		// Properties:
		IF (BACnet_Param.bStateText_WriteProtect) THEN
			WriteProtectProperty(E_BACnetPropIdentifier.PropActiveText, TRUE);
			WriteProtectProperty(E_BACnetPropIdentifier.PropInactiveText, TRUE);
		END_IF
		
		// Ensure UTF-8 Encoding:
		F_BA_EnsureUTF8(ADR(sDeviceType), SIZEOF(sDeviceType));
		F_BA_EnsureUTF8(ADR(sInactiveText), SIZEOF(sInactiveText));
		F_BA_EnsureUTF8(ADR(sActiveText), SIZEOF(sActiveText));

	TCOM_STATE.TCOM_STATE_SAFEOP:
		SyncPropertyPvPrio(E_BACnetPropIdentifier.PropPresentValue, SIZEOF(bValPgm), ADR(bValPgm), ADR(bEnPgm), BACnet_Param.ePrio_Program, 0, eFullSync_InitPLC, TRUE);
		
		SyncProperty(E_BACnetPropIdentifier.PropPresentValue, SIZEOF(bPresentValue), ADR(bPresentValue), 0, eSync_FromSupplement, TRUE);
		SyncProperty(E_BACnetPropIdentifier.PropCurrentlyActivePriority, SIZEOF(eActivePrio), ADR(eActivePrio), 0, eSync_FromSupplement, TRUE);
		
		SyncProperty(E_BACnetPropIdentifier.PropFeedbackValue, SIZEOF(_bFeedbackValue), ADR(_bFeedbackValue), 0, eSync_ToSupplement, TRUE);
		
	TCOM_STATE.TCOM_STATE_OP:
		SyncProperty(E_BACnetPropIdentifier.PropDeviceType, SIZEOF(sDeviceType), ADR(sDeviceType), 0, eFullSync_InitPLC, FALSE);
		SyncProperty(E_BACnetPropIdentifier.PropOutOfService, SIZEOF(bOutOfService), ADR(bOutOfService), 0, eFullSync_InitPLC, FALSE);
		SyncProperty(E_BACnetPropIdentifier.PropMinimumOffTime, SIZEOF(nMinimumOffTime), ADR(nMinimumOffTime), 0, eFullSync_InitPLC, FALSE);	
		SyncProperty(E_BACnetPropIdentifier.PropMinimumOnTime, SIZEOF(nMinimumOnTime), ADR(nMinimumOnTime), 0, eFullSync_InitPLC, FALSE);	
		SyncProperty(E_BACnetPropIdentifier.PropRelinquishDefault, SIZEOF(bRelinquishDefault), ADR(bRelinquishDefault), 0, eFullSync_InitPLC, FALSE);	
		SyncProperty(E_BACnetPropIdentifier.PropActiveText, SIZEOF(sActiveText), ADR(sActiveText), 0, eFullSync_InitPLC, FALSE);	
		SyncProperty(E_BACnetPropIdentifier.PropInactiveText, SIZEOF(sInactiveText), ADR(sInactiveText), 0, eFullSync_InitPLC, FALSE);
		SyncProperty(E_BACnetPropIdentifier.PropPolarity, SIZEOF(ePolarity), ADR(ePolarity), 0, eFullSync_InitPLC, FALSE);

		SyncProperty(E_BACnetPropIdentifier.PropChangeOfStateCount, SIZEOF(nChangeOfStateCount), ADR(nChangeOfStateCount), 0, eFullSync_InitPLC, FALSE);
		SyncProperty(E_BACnetPropIdentifier.PropChangeOfStateTime, SIZEOF(stChangeOfStateTime), ADR(stChangeOfStateTime), 0, eSync_FromSupplement, FALSE);
		SyncProperty(E_BACnetPropIdentifier.PropTimeOfStateCountReset, SIZEOF(stTimeOfStateCountReset), ADR(stTimeOfStateCountReset), 0, eSync_FromSupplement, FALSE);

		SyncProperty(E_BACnetPropIdentifier.PropElapsedActiveTime, SIZEOF(nElapsedActiveTime), ADR(nElapsedActiveTime), 0, eFullSync_InitPLC, FALSE);
		SyncProperty(E_BACnetPropIdentifier.PropTimeOfActiveTimeReset, SIZEOF(stTimeOfActiveTimeReset), ADR(stTimeOfActiveTimeReset), 0, eSync_FromSupplement, FALSE);
		
END_CASE
END_METHOD

METHOD FB_init : BOOL
VAR_INPUT
	bInitRetains : BOOL; // if TRUE, the retain variables are initialized (warm start / cold start)
	bInCopyCode : BOOL;  // if TRUE, the instance afterwards gets moved into the copy code (online change)
END_VAR
eObjectType := E_BACnetObjType.ObjBinaryOutput;
END_METHOD

PROPERTY ActivePrio : E_BACnet_Priority
GET
ActivePrio := eActivePrio;
END_GET
END_PROPERTY

PROPERTY ChangeOfStateTime : ST_BA_DateTime
GET
ChangeOfStateTime := stChangeOfStateTime;
END_GET
END_PROPERTY

PROPERTY TimeOfActiveTimeReset : ST_BA_DateTime
GET
TimeOfActiveTimeReset := stTimeOfActiveTimeReset;
END_GET
END_PROPERTY

PROPERTY TimeOfStateCountReset : ST_BA_DateTime
GET
TimeOfStateCountReset := stTimeOfStateCountReset;
END_GET
END_PROPERTY

END_FUNCTION_BLOCK

// POUs/Local/Objects/5P/FB_BACnet_BO_Raw5P
// Binary Output Object
// - Raw communication
// - 5 Priorities
{attribute 'pin_presentation_order_inputs' := 'bEnSfty,bValSfty,bEnCrit,bValCrit,bEnManLoc,bValManLoc,bEnPgm,bValPgm'}
{attribute 'pin_presentation_order_outputs' := 'bPresentValue,eActivePrio,bEvent,eReliability'}
{attribute 'enable_dynamic_creation'}
FUNCTION_BLOCK FB_BACnet_BO_Raw5P EXTENDS FB_BACnet_BO_Raw
VAR_INPUT
	bEnSfty					: BOOL;
	bValSfty				: BOOL;
	bEnCrit					: BOOL;
	bValCrit				: BOOL;
	bEnManLoc				: BOOL;
	bValManLoc				: BOOL;
END_VAR
VAR_INPUT CONSTANT PERSISTENT
	{region 'Operational Parameters'}
		{attribute 'parameterCategory':='Manual'}
		bEnManualRm : BOOL;
		{attribute 'parameterCategory':='Manual'}
		bValManualRm : BOOL;
	{endregion}
END_VAR

SUPER^();

METHOD PROTECTED OnObjectStateChanged
SUPER^.OnObjectStateChanged();

CASE (tState) OF
	TCOM_STATE.TCOM_STATE_PREOP:
		// SyncHandler:
		RequestSyncHandlers(1, 4);
		
	TCOM_STATE.TCOM_STATE_SAFEOP:
		SyncPropertyPvPrio(E_BACnetPropIdentifier.PropPresentValue, SIZEOF(bValSfty), ADR(bValSfty), ADR(bEnSfty), BACnet_Param.ePrio_LifeSafety, 0, eFullSync_InitPLC, TRUE);
		SyncPropertyPvPrio(E_BACnetPropIdentifier.PropPresentValue, SIZEOF(bValCrit), ADR(bValCrit), ADR(bEnCrit), BACnet_Param.ePrio_Critical, 0, eFullSync_InitPLC, TRUE);
		SyncPropertyPvPrio(E_BACnetPropIdentifier.PropPresentValue, SIZEOF(bValManLoc), ADR(bValManLoc), ADR(bEnManLoc), BACnet_Param.ePrio_ManLocal, 0, eFullSync_InitPLC, TRUE);
		SyncPropertyPvPrio(E_BACnetPropIdentifier.PropPresentValue, SIZEOF(bValManualRm), ADR(bValManualRm), ADR(bEnManualRm), BACnet_Param.ePrio_ManRemote, 0, eFullSync_InitPLC, TRUE);
		
	TCOM_STATE.TCOM_STATE_OP:
		;
		
END_CASE
END_METHOD

PROPERTY EnManualRm : BOOL
GET
EnManualRm := bEnManualRm;
END_GET
SET
bEnManualRm := EnManualRm;
END_SET
END_PROPERTY

PROPERTY ValManualRm : BOOL
GET
ValManualRm := bValManualRm;
END_GET
SET
bValManualRm := ValManualRm;
END_SET
END_PROPERTY

END_FUNCTION_BLOCK

// POUs/Local/Objects/FB_BACnet_BV
// Binary Value Object
// - 1 Priority
{attribute 'enable_dynamic_creation'}
FUNCTION_BLOCK FB_BACnet_BV EXTENDS FB_BACnet_EventObject
VAR_INPUT
	bEnPgm		: BOOL;
	bValPgm		: BOOL;
END_VAR
VAR_INPUT CONSTANT PERSISTENT
	{region 'Variable Parameters'}
		{attribute 'parameterCategory':='General'}
		{attribute 'parameterUnit':= 's'}
		nMinimumOffTime : UDINT;
		{attribute 'parameterCategory':='General'}
		{attribute 'parameterUnit':= 's'}
		nMinimumOnTime : UDINT;
		
		{attribute 'parameterCategory':='Value'}
		bRelinquishDefault : BOOL;
		{attribute 'parameterCategory':='Value'}
		bOutOfService : BOOL;
		{attribute 'parameterCategory':='Value'}
		{attribute 'TcEncoding':='UTF-8'}
		sInactiveText : T_BACnet_StateText;
		{attribute 'parameterCategory':='Value'}
		{attribute 'TcEncoding':='UTF-8'}
		sActiveText : T_BACnet_StateText;
		
		{attribute 'parameterCategory':='EventConfig'}
		bAlarmValue : BOOL := TRUE;
			 
		{attribute 'parameterCategory':='StateChange'}
		nChangeOfStateCount : UDINT;
		
		{attribute 'parameterCategory':='ActiveTime'}
		{attribute 'parameterUnit':= 's'}
		nElapsedActiveTime : UDINT;
	{endregion}
END_VAR
VAR_OUTPUT
	bPresentValue	: BOOL;
	eActivePrio		: E_BACnet_Priority;			// Indicates the currently active priority of the priority array
END_VAR
VAR
	{region 'Output-Properties'}
		{attribute 'parameterCategory':='StateChange'}
		stChangeOfStateTime : ST_BA_DateTime;
		{attribute 'parameterCategory':='StateChange'}
		stTimeOfStateCountReset : ST_BA_DateTime;
		
		{attribute 'parameterCategory':='ActiveTime'}
		stTimeOfActiveTimeReset : ST_BA_DateTime;
	{endregion}
END_VAR

SUPER^();

METHOD PROTECTED OnObjectStateChanged
SUPER^.OnObjectStateChanged();

CASE (tState) OF
	TCOM_STATE.TCOM_STATE_PREOP:
		// SyncHandler:
		RequestSyncHandlers(4, 10);
		
		// Properties:
		EnableProperty(E_BACnetPropIdentifier.PropDeviceType, FALSE);

		IF (BACnet_Param.bStateText_WriteProtect) THEN
			WriteProtectProperty(E_BACnetPropIdentifier.PropActiveText, TRUE);
			WriteProtectProperty(E_BACnetPropIdentifier.PropInactiveText, TRUE);
		END_IF
		
		// Ensure UTF-8 Encoding:
		F_BA_EnsureUTF8(ADR(sInactiveText), SIZEOF(sInactiveText));
		F_BA_EnsureUTF8(ADR(sActiveText), SIZEOF(sActiveText));

	TCOM_STATE.TCOM_STATE_SAFEOP:
		SyncPropertyPvPrio(E_BACnetPropIdentifier.PropPresentValue, SIZEOF(bValPgm), ADR(bValPgm), ADR(bEnPgm), BACnet_Param.ePrio_Program, 0, eFullSync_InitPLC, TRUE);
		
		SyncProperty(E_BACnetPropIdentifier.PropPresentValue, SIZEOF(bPresentValue), ADR(bPresentValue), 0, eSync_FromSupplement, TRUE);
		SyncProperty(E_BACnetPropIdentifier.PropCurrentlyActivePriority, SIZEOF(eActivePrio), ADR(eActivePrio), 0, eSync_FromSupplement, TRUE);
		
	TCOM_STATE.TCOM_STATE_OP:
		SyncProperty(E_BACnetPropIdentifier.PropAlarmValue, SIZEOF(bAlarmValue), ADR(bAlarmValue), 0, eFullSync_InitPLC, FALSE);
		SyncProperty(E_BACnetPropIdentifier.PropOutOfService, SIZEOF(bOutOfService), ADR(bOutOfService), 0, eFullSync_InitPLC, FALSE);
		SyncProperty(E_BACnetPropIdentifier.PropMinimumOffTime, SIZEOF(nMinimumOffTime), ADR(nMinimumOffTime), 0, eFullSync_InitPLC, FALSE);	
		SyncProperty(E_BACnetPropIdentifier.PropMinimumOnTime, SIZEOF(nMinimumOnTime), ADR(nMinimumOnTime), 0, eFullSync_InitPLC, FALSE);	
		SyncProperty(E_BACnetPropIdentifier.PropRelinquishDefault, SIZEOF(bRelinquishDefault), ADR(bRelinquishDefault), 0, eFullSync_InitPLC, FALSE);	
		SyncProperty(E_BACnetPropIdentifier.PropActiveText, SIZEOF(sActiveText), ADR(sActiveText), 0, eFullSync_InitPLC, FALSE);	
		SyncProperty(E_BACnetPropIdentifier.PropInactiveText, SIZEOF(sInactiveText), ADR(sInactiveText), 0, eFullSync_InitPLC, FALSE);

		SyncProperty(E_BACnetPropIdentifier.PropChangeOfStateCount, SIZEOF(nChangeOfStateCount), ADR(nChangeOfStateCount), 0, eFullSync_InitPLC, FALSE);
		SyncProperty(E_BACnetPropIdentifier.PropChangeOfStateTime, SIZEOF(stChangeOfStateTime), ADR(stChangeOfStateTime), 0, eSync_FromSupplement, FALSE);
		SyncProperty(E_BACnetPropIdentifier.PropTimeOfStateCountReset, SIZEOF(stTimeOfStateCountReset), ADR(stTimeOfStateCountReset), 0, eSync_FromSupplement, FALSE);

		SyncProperty(E_BACnetPropIdentifier.PropElapsedActiveTime, SIZEOF(nElapsedActiveTime), ADR(nElapsedActiveTime), 0, eFullSync_InitPLC, FALSE);
		SyncProperty(E_BACnetPropIdentifier.PropTimeOfActiveTimeReset, SIZEOF(stTimeOfActiveTimeReset), ADR(stTimeOfActiveTimeReset), 0, eSync_FromSupplement, FALSE);
		
END_CASE
END_METHOD

METHOD FB_init : BOOL
VAR_INPUT
	bInitRetains : BOOL; // if TRUE, the retain variables are initialized (warm start / cold start)
	bInCopyCode : BOOL;  // if TRUE, the instance afterwards gets moved into the copy code (online change)
END_VAR
eObjectType := E_BACnetObjType.ObjBinaryValue;
END_METHOD

PROPERTY ActivePrio : E_BACnet_Priority
GET
ActivePrio := eActivePrio;
END_GET
END_PROPERTY

PROPERTY ChangeOfStateTime : ST_BA_DateTime
GET
ChangeOfStateTime := stChangeOfStateTime;
END_GET
END_PROPERTY

PROPERTY TimeOfActiveTimeReset : ST_BA_DateTime
GET
TimeOfActiveTimeReset := stTimeOfActiveTimeReset;
END_GET
END_PROPERTY

PROPERTY TimeOfStateCountReset : ST_BA_DateTime
GET
TimeOfStateCountReset := stTimeOfStateCountReset;
END_GET
END_PROPERTY

END_FUNCTION_BLOCK

// POUs/Local/Objects/5P/FB_BACnet_BV_5P
// Binary Value Object
// - 5 Priorities
{attribute 'pin_presentation_order_inputs' := 'bEnSfty,bValSfty,bEnCrit,bValCrit,bEnManLoc,bValManLoc,bEnPgm,bValPgm'}
{attribute 'pin_presentation_order_outputs' := 'bPresentValue,eActivePrio,bEvent,eReliability'}
{attribute 'enable_dynamic_creation'}
FUNCTION_BLOCK FB_BACnet_BV_5P EXTENDS FB_BACnet_BV
VAR_INPUT
	bEnSfty					: BOOL;
	bValSfty				: BOOL;
	bEnCrit					: BOOL;
	bValCrit				: BOOL;
	bEnManLoc				: BOOL;
	bValManLoc				: BOOL;
END_VAR
VAR_INPUT CONSTANT PERSISTENT
	{region 'Operational Parameters'}
		{attribute 'parameterCategory':='Manual'}
		bEnManualRm : BOOL;
		{attribute 'parameterCategory':='Manual'}
		bValManualRm : BOOL;
	{endregion}
END_VAR

SUPER^();

METHOD PROTECTED OnObjectStateChanged
SUPER^.OnObjectStateChanged();

CASE (tState) OF
	TCOM_STATE.TCOM_STATE_PREOP:
		// SyncHandler:
		RequestSyncHandlers(1, 4);
		
	TCOM_STATE.TCOM_STATE_SAFEOP:
		SyncPropertyPvPrio(E_BACnetPropIdentifier.PropPresentValue, SIZEOF(bValSfty), ADR(bValSfty), ADR(bEnSfty), BACnet_Param.ePrio_LifeSafety, 0, eFullSync_InitPLC, TRUE);
		SyncPropertyPvPrio(E_BACnetPropIdentifier.PropPresentValue, SIZEOF(bValCrit), ADR(bValCrit), ADR(bEnCrit), BACnet_Param.ePrio_Critical, 0, eFullSync_InitPLC, TRUE);
		SyncPropertyPvPrio(E_BACnetPropIdentifier.PropPresentValue, SIZEOF(bValManLoc), ADR(bValManLoc), ADR(bEnManLoc), BACnet_Param.ePrio_ManLocal, 0, eFullSync_InitPLC, TRUE);
		SyncPropertyPvPrio(E_BACnetPropIdentifier.PropPresentValue, SIZEOF(bValManualRm), ADR(bValManualRm), ADR(bEnManualRm), BACnet_Param.ePrio_ManRemote, 0, eFullSync_InitPLC, TRUE);
		
	TCOM_STATE.TCOM_STATE_OP:
		;
		
END_CASE
END_METHOD

PROPERTY EnManualRm : BOOL
GET
EnManualRm := bEnManualRm;
END_GET
SET
bEnManualRm := EnManualRm;
END_SET
END_PROPERTY

PROPERTY ValManualRm : BOOL
GET
ValManualRm := bValManualRm;
END_GET
SET
bValManualRm := ValManualRm;
END_SET
END_PROPERTY

END_FUNCTION_BLOCK

// POUs/Local/Objects/FB_BACnet_BV_Disp
// Binary Setpoint Object for Operation
// - Used to display a value
{attribute 'enable_dynamic_creation'}
FUNCTION_BLOCK FB_BACnet_BV_Disp EXTENDS FB_BACnet_Object
VAR_INPUT
	bVal			: BOOL;
END_VAR
VAR_INPUT CONSTANT PERSISTENT
	{region 'Variable Parameters'}
		{attribute 'parameterCategory':='Value'}
		{attribute 'TcEncoding':='UTF-8'}
		sInactiveText : T_BACnet_StateText;
		{attribute 'parameterCategory':='Value'}
		{attribute 'TcEncoding':='UTF-8'}
		sActiveText : T_BACnet_StateText;
	{endregion}
END_VAR
VAR_OUTPUT
	bPresentValue	: BOOL;
END_VAR

IF bReady THEN
	bPresentValue := bVal;
ELSE
	bPresentValue := FALSE;
END_IF

SUPER^();

METHOD PROTECTED OnObjectStateChanged
SUPER^.OnObjectStateChanged();

CASE (tState) OF
	TCOM_STATE.TCOM_STATE_PREOP:
		// SyncHandler:
		RequestSyncHandlers(0, 3);
		
		// Properties:
		EnableProperty(E_BACnetPropIdentifier.PropDeviceType, FALSE);
		EnableProperty(E_BACnetPropIdentifier.PropMinimumOnTime, FALSE);
		EnableProperty(E_BACnetPropIdentifier.PropMinimumOffTime, FALSE);
		EnableProperty(E_BACnetPropIdentifier.PropNotificationClass, FALSE);
		EnableProperty(E_BACnetPropIdentifier.PropNotifyType, FALSE);
		EnableProperty(E_BACnetPropIdentifier.PropEventEnable, FALSE);
		EnableProperty(E_BACnetPropIdentifier.PropEventTimeStamps, FALSE);
		EnableProperty(E_BACnetPropIdentifier.PropEventMessageTexts, FALSE);
		EnableProperty(E_BACnetPropIdentifier.PropEventMessageTextsConfig, FALSE);
		EnableProperty(E_BACnetPropIdentifier.PropTimeDelay, FALSE);
		EnableProperty(E_BACnetPropIdentifier.PropAckedTransitions, FALSE);
		EnableProperty(E_BACnetPropIdentifier.PropReliability, FALSE);
		EnableProperty(E_BACnetPropIdentifier.PropEventDetectionEnable, FALSE);
		EnableProperty(E_BACnetPropIdentifier.PropEventAlgorithmInhibit, FALSE);
		EnableProperty(E_BACnetPropIdentifier.PropTimeDelayNormal, FALSE);
		EnableProperty(E_BACnetPropIdentifier.PropReliabilityEvaluationInhibit, FALSE);
		EnableProperty(E_BACnetPropIdentifier.PropChangeOfStateCount, FALSE);
		EnableProperty(E_BACnetPropIdentifier.PropChangeOfStateTime, FALSE);
		EnableProperty(E_BACnetPropIdentifier.PropTimeOfStateCountReset, FALSE);
		EnableProperty(E_BACnetPropIdentifier.PropElapsedActiveTime, FALSE);
		EnableProperty(E_BACnetPropIdentifier.PropTimeOfActiveTimeReset, FALSE);
		EnableProperty(E_BACnetPropIdentifier.PropRelinquishDefault, FALSE);
		EnableProperty(E_BACnetPropIdentifier.PropPriorityArray, FALSE);
		EnableProperty(E_BACnetPropIdentifier.PropCurrentlyActivePriority, FALSE);
		
		WriteProtectProperty(E_BACnetPropIdentifier.PropOutOfService, TRUE);
		// EnableProperty(E_BACnetPropIdentifier.PropStatusFlags, FALSE);
		// EnableProperty(E_BACnetPropIdentifier.PropEventState, FALSE);
		
		WriteProtectProperty(E_BACnetPropIdentifier.PropPresentValue, TRUE);
		
		IF (BACnet_Param.bStateText_WriteProtect) THEN
			WriteProtectProperty(E_BACnetPropIdentifier.PropActiveText, TRUE);
			WriteProtectProperty(E_BACnetPropIdentifier.PropInactiveText, TRUE);
		END_IF
		
		// Ensure UTF-8 Encoding:
		F_BA_EnsureUTF8(ADR(sInactiveText), SIZEOF(sInactiveText));
		F_BA_EnsureUTF8(ADR(sActiveText), SIZEOF(sActiveText));
		
	TCOM_STATE.TCOM_STATE_SAFEOP:
		SyncProperty(E_BACnetPropIdentifier.PropPresentValue, SIZEOF(bVal), ADR(bVal), 0, eSync_ToSupplement, TRUE);
		
	TCOM_STATE.TCOM_STATE_OP:
		SyncProperty(E_BACnetPropIdentifier.PropActiveText, SIZEOF(sActiveText), ADR(sActiveText), 0, eFullSync_InitPLC, FALSE);	
		SyncProperty(E_BACnetPropIdentifier.PropInactiveText, SIZEOF(sInactiveText), ADR(sInactiveText), 0, eFullSync_InitPLC, FALSE);
END_CASE
END_METHOD

METHOD FB_init : BOOL
VAR_INPUT
	bInitRetains : BOOL; // if TRUE, the retain variables are initialized (warm start / cold start)
	bInCopyCode : BOOL;  // if TRUE, the instance afterwards gets moved into the copy code (online change)
END_VAR
eObjectType := E_BACnetObjType.ObjBinaryValue;
END_METHOD

END_FUNCTION_BLOCK

// POUs/Local/Objects/FB_BACnet_BV_Setp
// Binary Setpoint Object for Operation
// - Used to define a setpoint by user
{attribute 'enable_dynamic_creation'}
FUNCTION_BLOCK FB_BACnet_BV_Setp EXTENDS FB_BACnet_Object
VAR_INPUT CONSTANT PERSISTENT
	{region 'Variable Parameters'}
		{attribute 'parameterCategory':='Value'}
		{attribute 'TcEncoding':='UTF-8'}
		sInactiveText : T_BACnet_StateText;
		{attribute 'parameterCategory':='Value'}
		{attribute 'TcEncoding':='UTF-8'}
		sActiveText : T_BACnet_StateText;
	{endregion}
	{region 'Operational Parameters'}
		{attribute 'parameterCategory':='Value'}
		bValue : BOOL;
	{endregion}
END_VAR
VAR_OUTPUT
	bPresentValue	: BOOL;
END_VAR

IF bReady THEN
	bPresentValue := bValue;
ELSE
	bPresentValue := FALSE;
END_IF

SUPER^();

METHOD PROTECTED OnObjectStateChanged
SUPER^.OnObjectStateChanged();

CASE (tState) OF
	TCOM_STATE.TCOM_STATE_PREOP:
		// SyncHandler:
		RequestSyncHandlers(0, 3);
		
		// Properties:
		EnableProperty(E_BACnetPropIdentifier.PropDeviceType, FALSE);
		EnableProperty(E_BACnetPropIdentifier.PropMinimumOnTime, FALSE);
		EnableProperty(E_BACnetPropIdentifier.PropMinimumOffTime, FALSE);
		EnableProperty(E_BACnetPropIdentifier.PropNotificationClass, FALSE);
		EnableProperty(E_BACnetPropIdentifier.PropNotifyType, FALSE);
		EnableProperty(E_BACnetPropIdentifier.PropEventEnable, FALSE);
		EnableProperty(E_BACnetPropIdentifier.PropEventTimeStamps, FALSE);
		EnableProperty(E_BACnetPropIdentifier.PropEventMessageTexts, FALSE);
		EnableProperty(E_BACnetPropIdentifier.PropEventMessageTextsConfig, FALSE);
		EnableProperty(E_BACnetPropIdentifier.PropTimeDelay, FALSE);
		EnableProperty(E_BACnetPropIdentifier.PropAckedTransitions, FALSE);
		EnableProperty(E_BACnetPropIdentifier.PropReliability, FALSE);
		EnableProperty(E_BACnetPropIdentifier.PropEventDetectionEnable, FALSE);
		EnableProperty(E_BACnetPropIdentifier.PropEventAlgorithmInhibit, FALSE);
		EnableProperty(E_BACnetPropIdentifier.PropTimeDelayNormal, FALSE);
		EnableProperty(E_BACnetPropIdentifier.PropReliabilityEvaluationInhibit, FALSE);
		EnableProperty(E_BACnetPropIdentifier.PropChangeOfStateCount, FALSE);
		EnableProperty(E_BACnetPropIdentifier.PropChangeOfStateTime, FALSE);
		EnableProperty(E_BACnetPropIdentifier.PropTimeOfStateCountReset, FALSE);
		EnableProperty(E_BACnetPropIdentifier.PropElapsedActiveTime, FALSE);
		EnableProperty(E_BACnetPropIdentifier.PropTimeOfActiveTimeReset, FALSE);
		EnableProperty(E_BACnetPropIdentifier.PropRelinquishDefault, FALSE);
		EnableProperty(E_BACnetPropIdentifier.PropPriorityArray, FALSE);
		EnableProperty(E_BACnetPropIdentifier.PropCurrentlyActivePriority, FALSE);
		
		WriteProtectProperty(E_BACnetPropIdentifier.PropOutOfService, TRUE);
		// EnableProperty(E_BACnetPropIdentifier.PropStatusFlags, FALSE);
		// EnableProperty(E_BACnetPropIdentifier.PropEventState, FALSE);
		
		IF (BACnet_Param.bStateText_WriteProtect) THEN
			WriteProtectProperty(E_BACnetPropIdentifier.PropActiveText, TRUE);
			WriteProtectProperty(E_BACnetPropIdentifier.PropInactiveText, TRUE);
		END_IF
		
		// Ensure UTF-8 Encoding:
		F_BA_EnsureUTF8(ADR(sInactiveText), SIZEOF(sInactiveText));
		F_BA_EnsureUTF8(ADR(sActiveText), SIZEOF(sActiveText));
		
	TCOM_STATE.TCOM_STATE_SAFEOP:
		;
		
	TCOM_STATE.TCOM_STATE_OP:
		SyncProperty(E_BACnetPropIdentifier.PropPresentValue, SIZEOF(bValue), ADR(bValue), 0, eFullSync_InitPLC, FALSE);
		
		SyncProperty(E_BACnetPropIdentifier.PropActiveText, SIZEOF(sActiveText), ADR(sActiveText), 0, eFullSync_InitPLC, FALSE);	
		SyncProperty(E_BACnetPropIdentifier.PropInactiveText, SIZEOF(sInactiveText), ADR(sInactiveText), 0, eFullSync_InitPLC, FALSE);
END_CASE
END_METHOD

METHOD FB_init : BOOL
VAR_INPUT
	bInitRetains : BOOL; // if TRUE, the retain variables are initialized (warm start / cold start)
	bInCopyCode : BOOL;  // if TRUE, the instance afterwards gets moved into the copy code (online change)
END_VAR
eObjectType := E_BACnetObjType.ObjBinaryValue;
END_METHOD

END_FUNCTION_BLOCK

// POUs/Local/Objects/FB_BACnet_MI_Raw
// Multistate Input Object
// - Raw communication
{attribute 'pin_presentation_order_outputs' := 'nPresentValue,bEvent,eReliability'}
{attribute 'enable_dynamic_creation'}
FUNCTION_BLOCK FB_BACnet_MI_Raw EXTENDS FB_BACnet_BaseMI
VAR_INPUT
	nRawValue					: UDINT;			// Raw value
END_VAR

IF bReady THEN
	nPresentValue := nRawValue;
ELSE
	nPresentValue := 1;
END_IF

SUPER^();

END_FUNCTION_BLOCK

// POUs/Local/Objects/[Base]/FB_BACnet_BaseMI
FUNCTION_BLOCK FB_BACnet_BaseMI EXTENDS FB_BACnet_EventObject
VAR_INPUT CONSTANT PERSISTENT
	{region 'Variable Parameters'}
		{attribute 'parameterCategory':='Value'}
		bOutOfService : BOOL;
		
		{attribute 'parameterCategory':='Hardware'}
		{attribute 'TcEncoding':='UTF-8'}
		sDeviceType : STRING;
	{endregion}
	{region 'Fixed Parameters'}
		{attribute 'parameterCategory':='Value'}
		{attribute 'TcEncoding':='UTF-8'}
		aStateText : T_BACnet_StateTextArray := BACnet_Param.sMultistate_DefaultStateText;
		
		{attribute 'parameterCategory':='EventConfig'}
		aAlarmValues : T_BACnet_MultistateValue;
		{attribute 'parameterCategory':='EventConfig'}
		aFaultValues : T_BACnet_MultistateValue;
	{endregion}
END_VAR
VAR_OUTPUT
	nPresentValue		: UDINT		:= 1;
END_VAR
VAR
	{region 'Output-Properties'}
		nStateCount		: UDINT;
	{endregion}
END_VAR

SUPER^();

METHOD PROTECTED OnObjectStateChanged
SUPER^.OnObjectStateChanged();

CASE (tState) OF
	TCOM_STATE.TCOM_STATE_PREOP:
		// SyncHandler:
		{warning disable C0196}
		nStateCount := F_BACnet_GetUsedStateText(aStateText);
		
		RequestSyncHandlers(0, nStateCount);								// Handlers for "E_BACnetPropIdentifier.PropStateText"
		RequestSyncHandlers(0, F_BACnet_GetUsedUDINT(aAlarmValues));		// Handlers for "E_BACnetPropIdentifier.PropAlarmValues"
		RequestSyncHandlers(0, F_BACnet_GetUsedUDINT(aFaultValues));		// Handlers for "E_BACnetPropIdentifier.PropFaultValues"
		RequestSyncHandlers(0, 3);											// Handlers for other properties
		{warning restore C0196}
		
		// Properties:
		WriteProtectProperty(E_BACnetPropIdentifier.PropNumberOfStates, TRUE);
		
		IF (BACnet_Param.bStateText_WriteProtect) THEN
			WriteProtectProperty(E_BACnetPropIdentifier.PropStateText, TRUE);
		END_IF
		
		// Ensure UTF-8 Encoding:
		F_BA_EnsureUTF8(ADR(sDeviceType), SIZEOF(sDeviceType));
		F_BA_EnsureUTF8Array(ADR(aStateText), SIZEOF(aStateText[1]), TO_DINT(BACnet_Param.nMultistate_StateCount));

	TCOM_STATE.TCOM_STATE_SAFEOP:
		SyncProperty(E_BACnetPropIdentifier.PropPresentValue, SIZEOF(nPresentValue), ADR(nPresentValue), 0, eSync_ToSupplement, TRUE);
			
	TCOM_STATE.TCOM_STATE_OP:
		// Init number of used states:
		SetNumberOfStates(nStateCount);
		
		SyncProperty(E_BACnetPropIdentifier.PropOutOfService, SIZEOF(bOutOfService), ADR(bOutOfService), 0, eFullSync_InitPLC, FALSE);
		SyncProperty(E_BACnetPropIdentifier.PropDeviceType, SIZEOF(sDeviceType), ADR(sDeviceType), 0, eFullSync_InitPLC, FALSE);
		SyncPropertyList(E_BACnetPropIdentifier.PropStateText, ADR(aStateText), SIZEOF(T_BACnet_StateText), nStateCount, eFullSync_InitPLC, FALSE);
		SyncPropertyList(E_BACnetPropIdentifier.PropAlarmValues, ADR(aAlarmValues), SIZEOF(UDINT), nStateCount, eFullSync_InitPLC, TRUE);
		SyncPropertyList(E_BACnetPropIdentifier.PropFaultValues, ADR(aFaultValues), SIZEOF(UDINT), nStateCount, eFullSync_InitPLC, TRUE);

END_CASE
END_METHOD

METHOD FB_init : BOOL
VAR_INPUT
	bInitRetains : BOOL; // if TRUE, the retain variables are initialized (warm start / cold start)
	bInCopyCode : BOOL;  // if TRUE, the instance afterwards gets moved into the copy code (online change)
END_VAR
eObjectType := E_BACnetObjType.ObjMultistateInput;
END_METHOD

PROPERTY StateCount : UDINT
GET
StateCount := nStateCount;
END_GET
END_PROPERTY

END_FUNCTION_BLOCK

// POUs/Helper/[internal]/String/F_BACnet_GetUsedStateText
{attribute 'hide'} // [Workaround] Not hidden when lib is included
FUNCTION INTERNAL F_BACnet_GetUsedStateText : UDINT
VAR_IN_OUT
	aArray				: ARRAY[*] OF T_BACnet_StateText;
END_VAR
VAR
	_nTemp				: DINT;
END_VAR

F_BACnet_GetUsedStateText := 0;

FOR _nTemp := LOWER_BOUND(aArray, 1) TO UPPER_BOUND(aArray, 1) DO
	IF LEN(aArray[_nTemp]) = 0 THEN
		EXIT;
	ELSE
		F_BACnet_GetUsedStateText := (F_BACnet_GetUsedStateText+1);
	END_IF
END_FOR

END_FUNCTION

// POUs/Helper/[internal]/String/F_BACnet_GetUsedUDINT
{attribute 'hide'} // [Workaround] Not hidden when lib is included
FUNCTION INTERNAL F_BACnet_GetUsedUDINT : UDINT
VAR_IN_OUT
	aArray				: ARRAY[*] OF UDINT;
END_VAR
VAR
	_nTemp				: DINT;
END_VAR

F_BACnet_GetUsedUDINT := 0;

FOR _nTemp := LOWER_BOUND(aArray, 1) TO UPPER_BOUND(aArray, 1) DO
	IF (aArray[_nTemp] = 0) THEN
		EXIT;
	ELSE
		F_BACnet_GetUsedUDINT := (F_BACnet_GetUsedUDINT+1);
	END_IF
END_FOR

END_FUNCTION

// POUs/Local/Objects/FB_BACnet_MO_Raw
// Multistate Output Object
// - Raw communication
// - 1 Priority
{attribute 'pin_presentation_order_outputs' := 'fPresentValue,bEvent,eReliability'}
{attribute 'enable_dynamic_creation'}
FUNCTION_BLOCK FB_BACnet_MO_Raw EXTENDS FB_BACnet_BaseMO
VAR_INPUT
	bEnFeedback					: BOOL;				// Enable of writing to Feedback Value (optional)
	nRawValFeedback				: UDINT;			// Raw feedback Value
END_VAR
VAR_OUTPUT
	nRawValue					: UDINT;			// Raw value
END_VAR

IF (bReady) THEN
	// Feedback Value:
	_nFeedbackValue := MAX(1, SEL(bEnFeedback, nPresentValue, nRawValFeedback));
	
	// Raw-IO Value:
	nRawValue := nPresentValue;
END_IF

SUPER^();

END_FUNCTION_BLOCK

// POUs/Local/Objects/[Base]/FB_BACnet_BaseMO
FUNCTION_BLOCK FB_BACnet_BaseMO EXTENDS FB_BACnet_EventObject
VAR_INPUT
	bEnPgm					: BOOL;
	nValPgm					: UDINT		:= 1;
END_VAR
VAR_INPUT CONSTANT PERSISTENT
	{region 'Variable Parameters'}
		{attribute 'parameterCategory':='Value'}
		nRelinquishDefault : UDINT := 1;
		{attribute 'parameterCategory':='Value'}
		bOutOfService : BOOL;
	
		{attribute 'parameterCategory':='Hardware'}
		{attribute 'TcEncoding':='UTF-8'}
		sDeviceType : STRING;
	{endregion}
	{region 'Fixed Parameters'}
		{attribute 'parameterCategory':='Value'}
		{attribute 'TcEncoding':='UTF-8'}
		sStateText : T_BACnet_StateTextArray := BACnet_Param.sMultistate_DefaultStateText;
	{endregion}
END_VAR
VAR_OUTPUT
	nPresentValue			: UDINT		:= 1;
	eActivePrio				: E_BACnet_Priority;			// Indicates the currently active priority of the priority array
END_VAR
VAR
	{region 'Output-Properties'}
		nStateCount			: UDINT;
	{endregion}
END_VAR
VAR
	{region 'Internal'}
		_nFeedbackValue		: UDINT;
	{endregion}
END_VAR

SUPER^();

METHOD PROTECTED OnObjectStateChanged
SUPER^.OnObjectStateChanged();

CASE (tState) OF
	TCOM_STATE.TCOM_STATE_PREOP:
		// SyncHandler:
		{warning disable C0196}
		nStateCount := F_BACnet_GetUsedStateText(sStateText);
		{warning restore C0196}
		
		RequestSyncHandlers(0, nStateCount);								// Handlers for "E_BACnetPropIdentifier.PropStateText"
		RequestSyncHandlers(1, 5);											// Handlers for other properties
		
		// Properties:
		WriteProtectProperty(E_BACnetPropIdentifier.PropNumberOfStates, TRUE);
		
		IF (BACnet_Param.bStateText_WriteProtect) THEN
			WriteProtectProperty(E_BACnetPropIdentifier.PropStateText, TRUE);
		END_IF
		
		// Ensure UTF-8 Encoding:
		F_BA_EnsureUTF8(ADR(sDeviceType), SIZEOF(sDeviceType));
		F_BA_EnsureUTF8Array(ADR(sStateText), SIZEOF(sStateText[1]), TO_DINT(BACnet_Param.nMultistate_StateCount));
		
	TCOM_STATE.TCOM_STATE_SAFEOP:
		SyncPropertyPvPrio(E_BACnetPropIdentifier.PropPresentValue, SIZEOF(nValPgm), ADR(nValPgm), ADR(bEnPgm), BACnet_Param.ePrio_Program, 0, eFullSync_InitPLC, TRUE);
		
		SyncProperty(E_BACnetPropIdentifier.PropPresentValue, SIZEOF(nPresentValue), ADR(nPresentValue), 0, eSync_FromSupplement, TRUE);
		SyncProperty(E_BACnetPropIdentifier.PropCurrentlyActivePriority, SIZEOF(eActivePrio), ADR(eActivePrio), 0, eSync_FromSupplement, TRUE);
		
		SyncProperty(E_BACnetPropIdentifier.PropFeedbackValue, SIZEOF(_nFeedbackValue), ADR(_nFeedbackValue), 0, eSync_ToSupplement, TRUE);
		
	TCOM_STATE.TCOM_STATE_OP:
		// Init number of used states:
		SetNumberOfStates(nStateCount);
		
		SyncProperty(E_BACnetPropIdentifier.PropDeviceType, SIZEOF(sDeviceType), ADR(sDeviceType), 0, eFullSync_InitPLC, FALSE);
		SyncProperty(E_BACnetPropIdentifier.PropRelinquishDefault, SIZEOF(nRelinquishDefault), ADR(nRelinquishDefault), 0, eFullSync_InitPLC, FALSE);
		SyncProperty(E_BACnetPropIdentifier.PropOutOfService, SIZEOF(bOutOfService), ADR(bOutOfService), 0, eFullSync_InitPLC, FALSE);
		SyncPropertyList(E_BACnetPropIdentifier.PropStateText, ADR(sStateText), SIZEOF(T_BACnet_StateText), nStateCount, eFullSync_InitPLC, FALSE);
		
END_CASE
END_METHOD

METHOD FB_init : BOOL
VAR_INPUT
	bInitRetains : BOOL; // if TRUE, the retain variables are initialized (warm start / cold start)
	bInCopyCode : BOOL;  // if TRUE, the instance afterwards gets moved into the copy code (online change)
END_VAR
eObjectType := E_BACnetObjType.ObjMultistateOutput;
END_METHOD

PROPERTY ActivePrio : E_BACnet_Priority
GET
ActivePrio := eActivePrio;
END_GET
END_PROPERTY

PROPERTY StateCount : UDINT
GET
StateCount := nStateCount;
END_GET
END_PROPERTY

END_FUNCTION_BLOCK

// POUs/Local/Objects/5P/FB_BACnet_MO_Raw5P
// Multistate Output Object
// - Raw communication
// - 5 Priorities
{attribute 'pin_presentation_order_inputs' := 'bEnSfty,nValSfty,bEnCrit,nValCrit,bEnManLoc,nValManLoc,bEnPgm,nValPgm'}
{attribute 'pin_presentation_order_outputs' := 'nPresentValue,eActivePrio,bEvent,eReliability'}
{attribute 'enable_dynamic_creation'}
FUNCTION_BLOCK FB_BACnet_MO_Raw5P EXTENDS FB_BACnet_MO_Raw
VAR_INPUT
	bEnSfty					: BOOL;
	nValSfty				: UDINT		:= 1;
	bEnCrit					: BOOL;
	nValCrit				: UDINT		:= 1;
	bEnManLoc				: BOOL;
	nValManLoc				: UDINT		:= 1;
END_VAR
VAR_INPUT CONSTANT PERSISTENT
	{region 'Operational Parameters'}
		{attribute 'parameterCategory':='Manual'}
		bEnManualRm : BOOL;
		{attribute 'parameterCategory':='Manual'}
		nValManualRm : UDINT := 1;
	{endregion}
END_VAR

SUPER^();

METHOD PROTECTED OnObjectStateChanged
SUPER^.OnObjectStateChanged();

CASE (tState) OF
	TCOM_STATE.TCOM_STATE_PREOP:
		// SyncHandler:
		RequestSyncHandlers(1, 4);
		
	TCOM_STATE.TCOM_STATE_SAFEOP:
		SyncPropertyPvPrio(E_BACnetPropIdentifier.PropPresentValue, SIZEOF(nValSfty), ADR(nValSfty), ADR(bEnSfty), BACnet_Param.ePrio_LifeSafety, 0, eFullSync_InitPLC, TRUE);
		SyncPropertyPvPrio(E_BACnetPropIdentifier.PropPresentValue, SIZEOF(nValCrit), ADR(nValCrit), ADR(bEnCrit), BACnet_Param.ePrio_Critical, 0, eFullSync_InitPLC, TRUE);
		SyncPropertyPvPrio(E_BACnetPropIdentifier.PropPresentValue, SIZEOF(nValManLoc), ADR(nValManLoc), ADR(bEnManLoc), BACnet_Param.ePrio_ManLocal, 0, eFullSync_InitPLC, TRUE);
		SyncPropertyPvPrio(E_BACnetPropIdentifier.PropPresentValue, SIZEOF(nValManualRm), ADR(nValManualRm), ADR(bEnManualRm), BACnet_Param.ePrio_ManRemote, 0, eFullSync_InitPLC, TRUE);
		
	TCOM_STATE.TCOM_STATE_OP:
		;
		
END_CASE
END_METHOD

PROPERTY EnManualRm : BOOL
GET
EnManualRm := bEnManualRm;
END_GET
SET
bEnManualRm := EnManualRm;
END_SET
END_PROPERTY

PROPERTY ValManualRm : UDINT
GET
ValManualRm := nValManualRm;
END_GET
SET
nValManualRm := ValManualRm;
END_SET
END_PROPERTY

END_FUNCTION_BLOCK

// POUs/Local/Objects/FB_BACnet_MV
// Multistate Value Object
// - 1 Priority
{attribute 'enable_dynamic_creation'}
FUNCTION_BLOCK FB_BACnet_MV EXTENDS FB_BACnet_EventObject
VAR_INPUT
	bEnPgm					: BOOL;
	nValPgm					: UDINT		:= 1;
END_VAR
VAR_INPUT CONSTANT PERSISTENT
	{region 'Fixed Parameters'}
		{attribute 'parameterCategory':='Value'}
		{attribute 'TcEncoding':='UTF-8'}
		sStateText : T_BACnet_StateTextArray := BACnet_Param.sMultistate_DefaultStateText;
		
		{attribute 'parameterCategory':='EventConfig'}
		aAlarmValues : T_BACnet_MultistateValue;
		{attribute 'parameterCategory':='EventConfig'}
		aFaultValues : T_BACnet_MultistateValue;
	{endregion}
	{region 'Variable Parameters'}
		{attribute 'parameterCategory':='Value'}
		nRelinquishDefault : UDINT := 1;
		{attribute 'parameterCategory':='Value'}
		bOutOfService : BOOL;
	{endregion}
END_VAR
VAR_OUTPUT
	nPresentValue			: UDINT		:= 1;
	eActivePrio				: E_BACnet_Priority;			// Indicates the currently active priority of the priority array
END_VAR
VAR
	{region 'Output-Properties'}
		nStateCount			: UDINT;
	{endregion}
END_VAR

SUPER^();

METHOD PROTECTED OnObjectStateChanged
SUPER^.OnObjectStateChanged();

CASE (tState) OF
	TCOM_STATE.TCOM_STATE_PREOP:
		// SyncHandler:
		{warning disable C0196}
		nStateCount := F_BACnet_GetUsedStateText(sStateText);
		
		RequestSyncHandlers(0, nStateCount);								// Handlers for "E_BACnetPropIdentifier.PropStateText"
		RequestSyncHandlers(0, F_BACnet_GetUsedUDINT(aAlarmValues));		// Handlers for "E_BACnetPropIdentifier.PropAlarmValues"
		RequestSyncHandlers(0, F_BACnet_GetUsedUDINT(aFaultValues));		// Handlers for "E_BACnetPropIdentifier.PropFaultValues"
		RequestSyncHandlers(1, 3);											// Handlers for other properties
		{warning restore C0196}
		
		// Properties:
		EnableProperty(E_BACnetPropIdentifier.PropDeviceType, FALSE);
		
		WriteProtectProperty(E_BACnetPropIdentifier.PropNumberOfStates, TRUE);
		
		IF (BACnet_Param.bStateText_WriteProtect) THEN
			WriteProtectProperty(E_BACnetPropIdentifier.PropStateText, TRUE);
		END_IF
		
		// Ensure UTF-8 Encoding:
		F_BA_EnsureUTF8Array(ADR(sStateText), SIZEOF(sStateText[1]), TO_DINT(BACnet_Param.nMultistate_StateCount));
		
	TCOM_STATE.TCOM_STATE_SAFEOP:
		SyncPropertyPvPrio(E_BACnetPropIdentifier.PropPresentValue, SIZEOF(nValPgm), ADR(nValPgm), ADR(bEnPgm), BACnet_Param.ePrio_Program, 0, eFullSync_InitPLC, TRUE);
		
		SyncProperty(E_BACnetPropIdentifier.PropPresentValue, SIZEOF(nPresentValue), ADR(nPresentValue), 0, eSync_FromSupplement, TRUE);
		SyncProperty(E_BACnetPropIdentifier.PropCurrentlyActivePriority, SIZEOF(eActivePrio), ADR(eActivePrio), 0, eSync_FromSupplement, TRUE);
		
	TCOM_STATE.TCOM_STATE_OP:
		// Init number of used states:
		SetNumberOfStates(nStateCount);
		
		SyncProperty(E_BACnetPropIdentifier.PropRelinquishDefault, SIZEOF(nRelinquishDefault), ADR(nRelinquishDefault), 0, eFullSync_InitPLC, FALSE);
		SyncProperty(E_BACnetPropIdentifier.PropOutOfService, SIZEOF(bOutOfService), ADR(bOutOfService), 0, eFullSync_InitPLC, FALSE);
		SyncPropertyList(E_BACnetPropIdentifier.PropStateText, ADR(sStateText), SIZEOF(T_BACnet_StateText), nStateCount, eFullSync_InitPLC, FALSE);
		SyncPropertyList(E_BACnetPropIdentifier.PropAlarmValues, ADR(aAlarmValues), SIZEOF(UDINT), nStateCount, eFullSync_InitPLC, TRUE);
		SyncPropertyList(E_BACnetPropIdentifier.PropFaultValues, ADR(aFaultValues), SIZEOF(UDINT), nStateCount, eFullSync_InitPLC, TRUE);
		
END_CASE
END_METHOD

METHOD FB_init : BOOL
VAR_INPUT
	bInitRetains : BOOL; // if TRUE, the retain variables are initialized (warm start / cold start)
	bInCopyCode : BOOL;  // if TRUE, the instance afterwards gets moved into the copy code (online change)
END_VAR
eObjectType := E_BACnetObjType.ObjMultistateValue;
END_METHOD

PROPERTY ActivePrio : E_BACnet_Priority
GET
ActivePrio := eActivePrio;
END_GET
END_PROPERTY

PROPERTY StateCount : UDINT
GET
StateCount := nStateCount;
END_GET
END_PROPERTY

END_FUNCTION_BLOCK

// POUs/Local/Objects/5P/FB_BACnet_MV_5P
// Multistate Value Object
// - 5 Priorities
{attribute 'pin_presentation_order_inputs' := 'bEnSfty,nValSfty,bEnCrit,nValCrit,bEnManLoc,nValManLoc,bEnPgm,nValPgm'}
{attribute 'pin_presentation_order_outputs' := 'nPresentValue,eActivePrio,bEvent,eReliability'}
{attribute 'enable_dynamic_creation'}
FUNCTION_BLOCK FB_BACnet_MV_5P EXTENDS FB_BACnet_MV
VAR_INPUT
	bEnSfty					: BOOL;
	nValSfty				: UDINT		:= 1;
	bEnCrit					: BOOL;
	nValCrit				: UDINT		:= 1;
	bEnManLoc				: BOOL;
	nValManLoc				: UDINT		:= 1;
END_VAR
VAR_INPUT CONSTANT PERSISTENT
	{region 'Operational Parameters'}
		{attribute 'parameterCategory':='Manual'}
		bEnManualRm : BOOL;
		{attribute 'parameterCategory':='Manual'}
		nValManualRm : UDINT := 1;
	{endregion}
END_VAR

SUPER^();

METHOD PROTECTED OnObjectStateChanged
SUPER^.OnObjectStateChanged();

CASE (tState) OF
	TCOM_STATE.TCOM_STATE_PREOP:
		// SyncHandler:
		RequestSyncHandlers(1, 4);
		
	TCOM_STATE.TCOM_STATE_SAFEOP:
		SyncPropertyPvPrio(E_BACnetPropIdentifier.PropPresentValue, SIZEOF(nValSfty), ADR(nValSfty), ADR(bEnSfty), BACnet_Param.ePrio_LifeSafety, 0, eFullSync_InitPLC, TRUE);
		SyncPropertyPvPrio(E_BACnetPropIdentifier.PropPresentValue, SIZEOF(nValCrit), ADR(nValCrit), ADR(bEnCrit), BACnet_Param.ePrio_Critical, 0, eFullSync_InitPLC, TRUE);
		SyncPropertyPvPrio(E_BACnetPropIdentifier.PropPresentValue, SIZEOF(nValManLoc), ADR(nValManLoc), ADR(bEnManLoc), BACnet_Param.ePrio_ManLocal, 0, eFullSync_InitPLC, TRUE);
		SyncPropertyPvPrio(E_BACnetPropIdentifier.PropPresentValue, SIZEOF(nValManualRm), ADR(nValManualRm), ADR(bEnManualRm), BACnet_Param.ePrio_ManRemote, 0, eFullSync_InitPLC, TRUE);
		
	TCOM_STATE.TCOM_STATE_OP:
		;
		
END_CASE
END_METHOD

PROPERTY EnManualRm : BOOL
GET
EnManualRm := bEnManualRm;
END_GET
SET
bEnManualRm := EnManualRm;
END_SET
END_PROPERTY

PROPERTY ValManualRm : UDINT
GET
ValManualRm := nValManualRm;
END_GET
SET
nValManualRm := ValManualRm;
END_SET
END_PROPERTY

END_FUNCTION_BLOCK

// POUs/Local/Objects/FB_BACnet_MV_Disp
// Multistate Setpoint Object for Setpoint
// - Used to display a value
{attribute 'enable_dynamic_creation'}
FUNCTION_BLOCK FB_BACnet_MV_Disp EXTENDS FB_BACnet_Object
VAR_INPUT
	nVal				: UDINT		:= 1;
END_VAR
VAR_INPUT CONSTANT PERSISTENT
	{region 'Fixed Parameters'}
		{attribute 'parameterCategory':='Value'}
		{attribute 'TcEncoding':='UTF-8'}
		sStateText : T_BACnet_StateTextArray := BACnet_Param.sMultistate_DefaultStateText;
	{endregion}
END_VAR
VAR_OUTPUT
	nPresentValue		: UDINT		:= 1;
END_VAR
VAR
	{region 'Output-Properties'}
		nStateCount		: UDINT;
	{endregion}
END_VAR

IF bReady THEN
	nPresentValue := nVal;
ELSE
	nPresentValue := 1;
END_IF

SUPER^();

METHOD PROTECTED OnObjectStateChanged
SUPER^.OnObjectStateChanged();

CASE (tState) OF
	TCOM_STATE.TCOM_STATE_PREOP:
		// SyncHandler:
		{warning disable C0196}
		nStateCount := F_BACnet_GetUsedStateText(sStateText);
		{warning restore C0196}
		
		RequestSyncHandlers(0, nStateCount);								// Handlers for "E_BACnetPropIdentifier.PropStateText"
		RequestSyncHandlers(0, 1);											// Handlers for other properties
		
		// Properties:
		WriteProtectProperty(E_BACnetPropIdentifier.PropPresentValue, TRUE);
		WriteProtectProperty(E_BACnetPropIdentifier.PropNumberOfStates, TRUE);
		
		IF (BACnet_Param.bStateText_WriteProtect) THEN
			WriteProtectProperty(E_BACnetPropIdentifier.PropStateText, TRUE);
		END_IF
		
		EnableProperty(E_BACnetPropIdentifier.PropDeviceType, FALSE);
		EnableProperty(E_BACnetPropIdentifier.PropNotificationClass, FALSE);
		EnableProperty(E_BACnetPropIdentifier.PropNotifyType, FALSE);
		EnableProperty(E_BACnetPropIdentifier.PropEventEnable, FALSE);
		EnableProperty(E_BACnetPropIdentifier.PropEventTimeStamps, FALSE);
		EnableProperty(E_BACnetPropIdentifier.PropEventMessageTexts, FALSE);
		EnableProperty(E_BACnetPropIdentifier.PropEventMessageTextsConfig, FALSE);
		EnableProperty(E_BACnetPropIdentifier.PropTimeDelay, FALSE);
		EnableProperty(E_BACnetPropIdentifier.PropAckedTransitions, FALSE);
		EnableProperty(E_BACnetPropIdentifier.PropReliability, FALSE);
		EnableProperty(E_BACnetPropIdentifier.PropEventDetectionEnable, FALSE);
		EnableProperty(E_BACnetPropIdentifier.PropEventAlgorithmInhibit, FALSE);
		EnableProperty(E_BACnetPropIdentifier.PropTimeDelayNormal, FALSE);
		EnableProperty(E_BACnetPropIdentifier.PropReliabilityEvaluationInhibit, FALSE);
		EnableProperty(E_BACnetPropIdentifier.PropAlarmValues, FALSE);
		EnableProperty(E_BACnetPropIdentifier.PropFaultValues, FALSE);
		EnableProperty(E_BACnetPropIdentifier.PropRelinquishDefault, FALSE);
		EnableProperty(E_BACnetPropIdentifier.PropPriorityArray, FALSE);
		EnableProperty(E_BACnetPropIdentifier.PropCurrentlyActivePriority, FALSE);
		
		WriteProtectProperty(E_BACnetPropIdentifier.PropOutOfService, TRUE);
		// EnableProperty(E_BACnetPropIdentifier.PropStatusFlags, FALSE);
		// EnableProperty(E_BACnetPropIdentifier.PropEventState, FALSE);
		
		// Ensure UTF-8 Encoding:
		F_BA_EnsureUTF8Array(ADR(sStateText), SIZEOF(sStateText[1]), TO_DINT(BACnet_Param.nMultistate_StateCount));
		
	TCOM_STATE.TCOM_STATE_SAFEOP:
		SyncProperty(E_BACnetPropIdentifier.PropPresentValue, SIZEOF(nVal), ADR(nVal), 0, eSync_ToSupplement, TRUE);
		
	TCOM_STATE.TCOM_STATE_OP:
		// Init number of used states:
		SetNumberOfStates(nStateCount);
		
		SyncPropertyList(E_BACnetPropIdentifier.PropStateText, ADR(sStateText), SIZEOF(T_BACnet_StateText), nStateCount, eFullSync_InitPLC, FALSE);

END_CASE
END_METHOD

METHOD FB_init : BOOL
VAR_INPUT
	bInitRetains : BOOL; // if TRUE, the retain variables are initialized (warm start / cold start)
	bInCopyCode : BOOL;  // if TRUE, the instance afterwards gets moved into the copy code (online change)
END_VAR
eObjectType := E_BACnetObjType.ObjMultistateValue;
END_METHOD

PROPERTY StateCount : UDINT
GET
StateCount := nStateCount;
END_GET
END_PROPERTY

END_FUNCTION_BLOCK

// POUs/Local/Objects/FB_BACnet_MV_Setp
// Multistate Setpoint Object for Setpoint
// - Used to define a setpoint by user
{attribute 'enable_dynamic_creation'}
FUNCTION_BLOCK FB_BACnet_MV_Setp EXTENDS FB_BACnet_Object
VAR_INPUT CONSTANT PERSISTENT
	{region 'Fixed Parameters'}
		{attribute 'parameterCategory':='Value'}
		{attribute 'TcEncoding':='UTF-8'}
		sStateText : T_BACnet_StateTextArray := BACnet_Param.sMultistate_DefaultStateText;
	{endregion}
	{region 'Operational Parameters'}
		{attribute 'parameterCategory':='Value'}
		nValue : UDINT := 1;
	{endregion}
END_VAR
VAR_OUTPUT
	nPresentValue		: UDINT		:= 1;
END_VAR
VAR
	{region 'Output-Properties'}
		nStateCount		: UDINT;
	{endregion}
END_VAR

IF bReady THEN
	nPresentValue := nValue;
ELSE
	nPresentValue := 1;
END_IF

SUPER^();

METHOD PROTECTED OnObjectStateChanged
SUPER^.OnObjectStateChanged();

CASE (tState) OF
	TCOM_STATE.TCOM_STATE_PREOP:
		// SyncHandler:
		{warning disable C0196}
		nStateCount := F_BACnet_GetUsedStateText(sStateText);
		{warning restore C0196}
		
		RequestSyncHandlers(0, nStateCount);								// Handlers for "E_BACnetPropIdentifier.PropStateText"
		RequestSyncHandlers(0, 1);											// Handlers for other properties
		
		// Properties:
		WriteProtectProperty(E_BACnetPropIdentifier.PropNumberOfStates, TRUE);
		
		IF (BACnet_Param.bStateText_WriteProtect) THEN
			WriteProtectProperty(E_BACnetPropIdentifier.PropStateText, TRUE);
		END_IF
		
		EnableProperty(E_BACnetPropIdentifier.PropDeviceType, FALSE);
		EnableProperty(E_BACnetPropIdentifier.PropNotificationClass, FALSE);
		EnableProperty(E_BACnetPropIdentifier.PropNotifyType, FALSE);
		EnableProperty(E_BACnetPropIdentifier.PropEventEnable, FALSE);
		EnableProperty(E_BACnetPropIdentifier.PropEventTimeStamps, FALSE);
		EnableProperty(E_BACnetPropIdentifier.PropEventMessageTexts, FALSE);
		EnableProperty(E_BACnetPropIdentifier.PropEventMessageTextsConfig, FALSE);
		EnableProperty(E_BACnetPropIdentifier.PropTimeDelay, FALSE);
		EnableProperty(E_BACnetPropIdentifier.PropAckedTransitions, FALSE);
		EnableProperty(E_BACnetPropIdentifier.PropReliability, FALSE);
		EnableProperty(E_BACnetPropIdentifier.PropEventDetectionEnable, FALSE);
		EnableProperty(E_BACnetPropIdentifier.PropEventAlgorithmInhibit, FALSE);
		EnableProperty(E_BACnetPropIdentifier.PropTimeDelayNormal, FALSE);
		EnableProperty(E_BACnetPropIdentifier.PropReliabilityEvaluationInhibit, FALSE);
		EnableProperty(E_BACnetPropIdentifier.PropAlarmValues, FALSE);
		EnableProperty(E_BACnetPropIdentifier.PropFaultValues, FALSE);
		EnableProperty(E_BACnetPropIdentifier.PropRelinquishDefault, FALSE);
		EnableProperty(E_BACnetPropIdentifier.PropPriorityArray, FALSE);
		EnableProperty(E_BACnetPropIdentifier.PropCurrentlyActivePriority, FALSE);
		
		WriteProtectProperty(E_BACnetPropIdentifier.PropOutOfService, TRUE);
		// EnableProperty(E_BACnetPropIdentifier.PropStatusFlags, FALSE);
		// EnableProperty(E_BACnetPropIdentifier.PropEventState, FALSE);
		
		// Ensure UTF-8 Encoding:
		F_BA_EnsureUTF8Array(ADR(sStateText), SIZEOF(sStateText[1]), TO_DINT(BACnet_Param.nMultistate_StateCount));
		
	TCOM_STATE.TCOM_STATE_SAFEOP:
		;
		
	TCOM_STATE.TCOM_STATE_OP:
		// Init number of used states:
		SetNumberOfStates(nStateCount);
		
		SyncProperty(E_BACnetPropIdentifier.PropPresentValue, SIZEOF(nValue), ADR(nValue), 0, eFullSync_InitPLC, FALSE);
		
		SyncPropertyList(E_BACnetPropIdentifier.PropStateText, ADR(sStateText), SIZEOF(T_BACnet_StateText), nStateCount, eFullSync_InitPLC, FALSE);

END_CASE
END_METHOD

METHOD FB_init : BOOL
VAR_INPUT
	bInitRetains : BOOL; // if TRUE, the retain variables are initialized (warm start / cold start)
	bInCopyCode : BOOL;  // if TRUE, the instance afterwards gets moved into the copy code (online change)
END_VAR
eObjectType := E_BACnetObjType.ObjMultistateValue;
END_METHOD

PROPERTY StateCount : UDINT
GET
StateCount := nStateCount;
END_GET
END_PROPERTY

END_FUNCTION_BLOCK

// POUs/Local/Objects/FB_BACnet_Cal
// Calendar Object
{attribute 'enable_dynamic_creation'}
FUNCTION_BLOCK FB_BACnet_Cal EXTENDS FB_BACnet_Object IMPLEMENTS I_BACnet_Cal
VAR_INPUT CONSTANT PERSISTENT
	{region 'Variable Parameters'}
		{attribute 'parameterCategory':='Value'}
		aDateList : T_BACnet_CalendarDateList;
	{endregion}
END_VAR
VAR_INPUT CONSTANT
	{region 'Variable Parameters'}
		{attribute 'parameterCategory':='Value'}
		bWriteDateList : BOOL;
	{endregion}
END_VAR
VAR_OUTPUT
	bPresentValue			: BOOL;
END_VAR
VAR	
	{region 'COV'}
		bDateListChanged	: BOOL;
	{endregion}
END_VAR

IF (bWriteDateList) THEN
	WriteContent();
	bWriteDateList := FALSE;
END_IF
IF (bDateListChanged) THEN
	ReadContent();
	bDateListChanged := FALSE;
END_IF

SUPER^();

METHOD PROTECTED OnObjectStateChanged
SUPER^.OnObjectStateChanged();

CASE (tState) OF
	TCOM_STATE.TCOM_STATE_PREOP:
		// SyncHandler:
		RequestSyncHandlers(2, 0);

	TCOM_STATE.TCOM_STATE_SAFEOP:
		;
		
	TCOM_STATE.TCOM_STATE_OP:
		SyncProperty(E_BACnetPropIdentifier.PropPresentValue, SIZEOF(bPresentValue), ADR(bPresentValue), 0, eSync_FromSupplement, FALSE);
		
		SyncPropertyCOV(E_BACnetPropIdentifier.PropDateList, ADR(bDateListChanged));
	
		WriteContent();
		
END_CASE
END_METHOD

METHOD FB_init : BOOL
VAR_INPUT
	bInitRetains : BOOL; // if TRUE, the retain variables are initialized (warm start / cold start)
	bInCopyCode : BOOL;  // if TRUE, the instance afterwards gets moved into the copy code (online change)
END_VAR
eObjectType := E_BACnetObjType.ObjCalendar;
END_METHOD

METHOD ReadContent : BOOL
ReadContent := (ReadPropertyDateList(aDateList) = S_OK);
END_METHOD

METHOD WriteContent : BOOL
WriteContent := (WritePropertyDateList(aDateList) = S_OK);
END_METHOD

END_FUNCTION_BLOCK

// POUs/Local/Objects/FB_BACnet_Device
// Device Object
{attribute 'enable_dynamic_creation'}
FUNCTION_BLOCK FB_BACnet_Device EXTENDS FB_BACnet_Object
VAR_INPUT CONSTANT PERSISTENT
	{region 'Variable Parameters'}
		{attribute 'parameterCategory':='Communication'}
		{attribute 'parameterUnit':= 'ms'}
		nAPDUSegmentTimeout : UDINT := 2000;						// (in [ms])
		{attribute 'parameterCategory':='Communication'}
		{attribute 'parameterUnit':= 'ms'}
		nAPDUTimeout : UDINT := 3000;								// (in [ms])
		{attribute 'parameterCategory':='Communication'}
		nNumberOfAPDURetries : UDINT := 3;
			 
		{attribute 'parameterCategory':='General'}
		{attribute 'TcEncoding':='UTF-8'}
		sLocation : T_MaxString;
	{endregion}
END_VAR
VAR_OUTPUT
	dtLocalTime			: ST_BA_DateTime;
END_VAR

SUPER^();

METHOD PROTECTED OnObjectStateChanged
SUPER^.OnObjectStateChanged();

CASE (tState) OF
	TCOM_STATE.TCOM_STATE_PREOP:
		// SyncHandler:
		RequestSyncHandlers(2, 4);
		
		// Ensure UTF-8 Encoding:
		F_BA_EnsureUTF8(ADR(sLocation), SIZEOF(sLocation));
		
	TCOM_STATE.TCOM_STATE_SAFEOP:
		;
	
	TCOM_STATE.TCOM_STATE_OP:
		SyncProperty(E_BACnetPropIdentifier.PropLocalTime, SIZEOF(dtLocalTime.stTime), ADR(dtLocalTime.stTime), 0, eSync_FromSupplement, FALSE);
		SyncProperty(E_BACnetPropIdentifier.PropLocalDate, SIZEOF(dtLocalTime.stDate), ADR(dtLocalTime.stDate), 0, eSync_FromSupplement, FALSE);
		
		SyncProperty(E_BACnetPropIdentifier.PropApduSegmentTimeout, SIZEOF(nAPDUSegmentTimeout), ADR(nAPDUSegmentTimeout), 0, eFullSync_InitPLC, FALSE);
		SyncProperty(E_BACnetPropIdentifier.PropApduTimeout, SIZEOF(nAPDUTimeout), ADR(nAPDUTimeout), 0, eFullSync_InitPLC, FALSE);
		SyncProperty(E_BACnetPropIdentifier.PropNumberOfAPDURetries, SIZEOF(nNumberOfAPDURetries), ADR(nNumberOfAPDURetries), 0, eFullSync_InitPLC, FALSE);
		SyncProperty(E_BACnetPropIdentifier.PropLocation, SIZEOF(sLocation), ADR(sLocation), 0, eFullSync_InitPLC, FALSE);
		
END_CASE
END_METHOD

METHOD FB_init : BOOL
VAR_INPUT
	bInitRetains : BOOL; // if TRUE, the retain variables are initialized (warm start / cold start)
	bInCopyCode : BOOL;  // if TRUE, the instance afterwards gets moved into the copy code (online change)
END_VAR
eObjectType := E_BACnetObjType.ObjDevice;
END_METHOD

PROPERTY Location : T_MaxString
GET
Location:=sLocation;
END_GET
SET
sLocation:=Location;
END_SET
END_PROPERTY

END_FUNCTION_BLOCK

// POUs/Local/Objects/FB_BACnet_File
// File Object
{attribute 'enable_dynamic_creation'}
FUNCTION_BLOCK FB_BACnet_File EXTENDS FB_BACnet_Object
VAR_INPUT CONSTANT
	{region 'Fixed Parameters'}
		{attribute 'parameterCategory':='General'}
		{attribute 'TcEncoding':='UTF-8'}
		sFileName : T_MaxString;
		{attribute 'parameterCategory':='General'}
		bEnBackupFile : BOOL;
	{endregion}
END_VAR
VAR_OUTPUT
	nFileSize		: UDINT;
END_VAR

SUPER^();

METHOD PROTECTED OnObjectStateChanged
SUPER^.OnObjectStateChanged();

CASE (tState) OF
	TCOM_STATE.TCOM_STATE_PREOP:
		// SyncHandler:
		IF sFileName <> '' THEN
			RequestSyncHandlers(1, 1);
			WritePropertyString(E_BACnetPropIdentifier.PropFileName, sFileName);
			EnableProperty(E_BACnetPropIdentifier.PropFileName, TRUE);
			WriteProtectProperty(E_BACnetPropIdentifier.PropFileName, TRUE);		
		ELSE
			RequestSyncHandlers(1, 0);
		END_IF
		IF bEnBackupFile THEN
			WritePropertyString(E_BACnetPropIdentifier.PropFileType, 'TwinCAT Configuration File');
		END_IF
		
	TCOM_STATE.TCOM_STATE_SAFEOP:
		;
	
	TCOM_STATE.TCOM_STATE_OP:
		SyncProperty(E_BACnetPropIdentifier.PropFileSize, SIZEOF(nFileSize), ADR(nFileSize), 0, eSync_FromSupplement, FALSE);
		IF sFileName <> '' THEN
			SyncProperty(E_BACnetPropIdentifier.PropFileName, SIZEOF(sFileName), ADR(sFileName), 0, eSync_ToSupplement, FALSE);
		END_IF
END_CASE
END_METHOD

METHOD FB_init : BOOL
VAR_INPUT
	bInitRetains : BOOL; // if TRUE, the retain variables are initialized (warm start / cold start)
	bInCopyCode : BOOL;  // if TRUE, the instance afterwards gets moved into the copy code (online change)
END_VAR
eObjectType := E_BACnetObjType.ObjFile;
END_METHOD

END_FUNCTION_BLOCK

// POUs/Local/Objects/FB_BACnet_Loop
// Loop Object
{attribute 'enable_dynamic_creation'}
FUNCTION_BLOCK FB_BACnet_Loop EXTENDS FB_BACnet_EventObject
VAR_INPUT
	bEn						: BOOL;
	fSetpoint				: REAL;
	fCtrlVar				: REAL;
END_VAR
VAR_INPUT CONSTANT PERSISTENT
	{region 'Variable Parameters'}
		{attribute 'parameterCategory':='Value'}
		bOutOfService : BOOL;
		{attribute 'parameterCategory':='Value'}
		fCOVIncrement : REAL := 0.1;
		{attribute 'parameterCategory':='Value'}
		eOutputUnit : E_BA_Unit := E_BA_Unit.eOther_Percent;
		
		{attribute 'parameterCategory':='Config'}
		eAction : E_BA_Action := E_BA_Action.eDirect;
		{attribute 'parameterCategory':='Config'}
		fBias : REAL := 0;
		{attribute 'parameterCategory':='Config'}
		fMinOutput : REAL := 0;
		{attribute 'parameterCategory':='Config'}
		fMaxOutput : REAL := 100;
		{attribute 'parameterCategory':='Config'}
		fAccLimit : REAL := 0.0;							// Setpoint acceleration limit positive and negative [1/s]
		{attribute 'parameterCategory':='Config'}
		fPropertionalConstant : REAL := 1;
		{attribute 'parameterCategory':='Config'}
		ePropertionalConstantUnit : E_BA_Unit := E_BA_Unit.eOther_NoUnits;
		{attribute 'parameterCategory':='Config'}
		fIntegralConstant : REAL := 60;
		{attribute 'parameterCategory':='Config'}
		eIntegralConstantUnit : E_BA_Unit := E_BA_Unit.eTime_Seconds;
		{attribute 'parameterCategory':='Config'}
		fDerivativeConstant : REAL := 0;
		{attribute 'parameterCategory':='Config'}
		eDerivativeConstantUnit : E_BA_Unit := E_BA_Unit.eTime_Seconds;
		
		{attribute 'parameterCategory':='EventConfig'}
		fDeadband : REAL := 0.1;
		{attribute 'parameterCategory':='EventConfig'}
		fErrorLimit : REAL := 0;
	{endregion}
END_VAR
VAR_OUTPUT
	fPresentValue			: REAL;
END_VAR
VAR
	{region 'Output-Properties'}
		eMode				: E_BACnet_LoopMode;
		fPropBand			: REAL; 						// Controller output in range of -100...100% in relation to Min.-/Max.-output
	{endregion}
END_VAR
VAR
	{region 'Internal'}
		{attribute 'hide'}
		fbIntCtrl			: FB_BACnet_PidControl;
		{attribute 'hide'}
		fbAccLimit			: FB_BACnet_AccLimit;
	{endregion}
	{region 'Temporary'}
		{attribute 'hide'}
		_sysTime			: GETCPUCOUNTER;
		{attribute 'hide'}
		_Time				: T_LARGE_INTEGER;
		{attribute 'hide'}
		_TimeOld			: T_LARGE_INTEGER;
		{attribute 'hide'}
		_tCycleTime			: REAL;
	{endregion}
END_VAR

IF (bReady) THEN
	// Determine cycle time:
	_TimeOld := _Time;
	_sysTime(cpuCntLoDW=>_Time.dwLowPart, cpuCntHiDW=>_Time.dwHighPart);
	_tCycleTime := F_BACnet_SysTimeDiff(In1:=_Time, In2:=_TimeOld);

	// Check PID mode:
	IF ((eIntegralConstantUnit = E_BA_Unit.eTime_Seconds OR eIntegralConstantUnit = 0) AND (eDerivativeConstantUnit = E_BA_Unit.eTime_Seconds)) AND
		((eDerivativeConstantUnit = E_BA_Unit.eTime_Seconds OR eDerivativeConstantUnit = 0) AND (eIntegralConstantUnit = E_BA_Unit.eTime_Seconds)) AND
		(ePropertionalConstantUnit = E_BA_Unit.eOther_NoUnits) THEN
		// Both are time_seconds:
		eMode := E_BACnet_LoopMode.eStandard;
		
	ELSIF (eIntegralConstantUnit <> E_BA_Unit.eTime_Seconds) AND
		(eDerivativeConstantUnit <> E_BA_Unit.eTime_Seconds) AND
		(ePropertionalConstantUnit = E_BA_Unit.eOther_NoUnits) THEN
		// Both are not time_seconds:
		eMode := E_BACnet_LoopMode.eIdeal;
		
	ELSE
		// Unknown settings - stop controller:
		eMode := E_BACnet_LoopMode.eNone;
	END_IF

	IF (NOT bEn) THEN
		fbIntCtrl.bReset := TRUE;
		
	ELSIF (eReliability <> E_BA_Reliability.eNoFaultDetected) OR (eMode = E_BACnet_LoopMode.eNone) THEN
		fbIntCtrl.bReset := TRUE;

	ELSIF stStatusFlags.bOutOfService THEN
		fbIntCtrl.bReset := TRUE;

	// Decide the control action (direct or reverse):
	ELSIF (eAction = E_BA_Action.eDirect) THEN
		fbIntCtrl.bReset := FALSE;
		fbIntCtrl.fPresentValue := fCtrlVar;
		fbIntCtrl.fSetpoint := fSetpoint;

	ELSIF (eAction = E_BA_Action.eReverse) THEN
		fbIntCtrl.bReset := FALSE;
		fbIntCtrl.fPresentValue := fSetpoint;
		fbIntCtrl.fSetpoint := fCtrlVar;

	ELSE
		// Unknown action:
		fbIntCtrl.bReset := TRUE;
	END_IF

	// Set parameter depending on mode:
	CASE eMode OF
		E_BACnet_LoopMode.eIdeal:
			fbIntCtrl.fKp := fPropertionalConstant;
			fbIntCtrl.fKi := fIntegralConstant;
			fbIntCtrl.fKd := fDerivativeConstant;
			
		E_BACnet_LoopMode.eStandard:
			// Kp = Kp:
			fbIntCtrl.fKp := fPropertionalConstant;
			
			// Ki = Kp / Ti:
			IF (fIntegralConstant <> 0.0) THEN
				fbIntCtrl.fKi := (fPropertionalConstant / fIntegralConstant);
			ELSE
				fbIntCtrl.fKi := 0.0;
			END_IF
			
			// Kd = Kp * Td:
			fbIntCtrl.fKd := (fPropertionalConstant * fDerivativeConstant);
			
	END_CASE

	// Call PID control function block:
	fbIntCtrl(
		fCtrlCycleTime := _tCycleTime,
		fBias := fBias,
		fTp := -1.0,
		fMinOutput := fMinOutput,
		fMaxOutput := fMaxOutput,
		fY => fbAccLimit.X
	);
END_IF

// Limit present value:
fbAccLimit(X:=fbIntCtrl.fY, Amax:=fAccLimit, Tcycle:=_tCycleTime, Y=>fPresentValue);

// Calculate proportional band:
IF (fMaxOutput > 0.0) AND (fMinOutput >= 0.0) THEN
	fPropBand := ((fPresentValue - fMinOutput) / (fMaxOutput - fMinOutput)) * 100.0;
ELSIF (fMaxOutput <= 0.0) AND (fMinOutput < 0.0) THEN
	fPropBand := ((fPresentValue - fMaxOutput) / (fMaxOutput - fMinOutput)) * 100.0;
ELSIF (fPresentValue > 0.0) AND (fMaxOutput > 0.0) THEN
	fPropBand := (fPresentValue / fMaxOutput) * 100.0;
ELSIF (fPresentValue < 0.0) AND (fMinOutput < 0.0) THEN
	fPropBand := (fPresentValue / fMinOutput) * -100.0;
ELSE
	fPropBand := 0.0;
END_IF

SUPER^();

METHOD PROTECTED OnObjectStateChanged
SUPER^.OnObjectStateChanged();

CASE (tState) OF
	TCOM_STATE.TCOM_STATE_PREOP:
		// SyncHandler:
		RequestSyncHandlers(0, 18);
		
		// Properties:
		EnableProperty(E_BACnetPropIdentifier.PropManipulatedVariableReference, FALSE);
		EnableProperty(E_BACnetPropIdentifier.PropControlledVariableReference, FALSE);
		EnableProperty(E_BACnetPropIdentifier.PropSetpointReference, FALSE);
		EnableProperty(E_BACnetPropIdentifier.PropControlledVariableUnits, FALSE);
		EnableProperty(E_BACnetPropIdentifier.PropUpdateInterval, FALSE);
		
		EnableProperty(E_BACnetPropIdentifier.PropPriorityForWriting, FALSE);
		
		WriteProtectProperty(E_BACnetPropIdentifier.PropPresentValue, TRUE);
		WriteProtectProperty(E_BACnetPropIdentifier.PropSetpoint, TRUE);
		WriteProtectProperty(E_BACnetPropIdentifier.PropControlledVariableValue, TRUE);
		
	TCOM_STATE.TCOM_STATE_SAFEOP:
		SyncProperty(E_BACnetPropIdentifier.PropPresentValue, SIZEOF(fPresentValue), ADR(fPresentValue), 0, eSync_ToSupplement, TRUE);
		SyncProperty(E_BACnetPropIdentifier.PropSetpoint, SIZEOF(fSetpoint), ADR(fSetpoint), 0, eSync_ToSupplement, TRUE);
		SyncProperty(E_BACnetPropIdentifier.PropControlledVariableValue, SIZEOF(fCtrlVar), ADR(fCtrlVar), 0, eSync_ToSupplement, TRUE);
	
	TCOM_STATE.TCOM_STATE_OP:
		SyncProperty(E_BACnetPropIdentifier.PropOutputUnits, SIZEOF(eOutputUnit), ADR(eOutputUnit), 0, eFullSync_InitPLC, FALSE);
		SyncProperty(E_BACnetPropIdentifier.PropOutOfService, SIZEOF(bOutOfService), ADR(bOutOfService), 0, eFullSync_InitPLC, FALSE);
		SyncProperty(E_BACnetPropIdentifier.PropCovIncrement, SIZEOF(fCOVIncrement), ADR(fCOVIncrement), 0, eFullSync_InitPLC, FALSE);
		SyncProperty(E_BACnetPropIdentifier.PropProportionalConstant, SIZEOF(fPropertionalConstant), ADR(fPropertionalConstant), 0, eFullSync_InitPLC, FALSE);
		SyncProperty(E_BACnetPropIdentifier.PropProportionalConstantUnits, SIZEOF(ePropertionalConstantUnit), ADR(ePropertionalConstantUnit), 0, eFullSync_InitPLC, FALSE);
		SyncProperty(E_BACnetPropIdentifier.PropIntegralConstant, SIZEOF(fIntegralConstant), ADR(fIntegralConstant), 0, eFullSync_InitPLC, FALSE);
		SyncProperty(E_BACnetPropIdentifier.PropIntegralConstantUnits, SIZEOF(eIntegralConstantUnit), ADR(eIntegralConstantUnit), 0, eFullSync_InitPLC, FALSE);
		SyncProperty(E_BACnetPropIdentifier.PropDerivativeConstant, SIZEOF(fDerivativeConstant), ADR(fDerivativeConstant), 0, eFullSync_InitPLC, FALSE);
		SyncProperty(E_BACnetPropIdentifier.PropDerivativeConstantUnits, SIZEOF(eDerivativeConstantUnit), ADR(eDerivativeConstantUnit), 0, eFullSync_InitPLC, FALSE);
		SyncProperty(E_BACnetPropIdentifier.PropDeadband, SIZEOF(fDeadband), ADR(fDeadband), 0, eFullSync_InitPLC, FALSE);
		SyncProperty(E_BACnetPropIdentifier.PropErrorLimit, SIZEOF(fErrorLimit), ADR(fErrorLimit), 0, eFullSync_InitPLC, FALSE);
		SyncProperty(E_BACnetPropIdentifier.PropMinimumOutput, SIZEOF(fMinOutput), ADR(fMinOutput), 0, eFullSync_InitPLC, FALSE);
		SyncProperty(E_BACnetPropIdentifier.PropMaximumOutput, SIZEOF(fMaxOutput), ADR(fMaxOutput), 0, eFullSync_InitPLC, FALSE);
		SyncProperty(E_BACnetPropIdentifier.PropActionProp, SIZEOF(eAction), ADR(eAction), 0, eFullSync_InitPLC, FALSE);
		SyncProperty(E_BACnetPropIdentifier.PropBias, SIZEOF(fBias), ADR(fBias), 0, eFullSync_InitPLC, FALSE);
		
END_CASE
END_METHOD

METHOD FB_init : BOOL
VAR_INPUT
	bInitRetains : BOOL; // if TRUE, the retain variables are initialized (warm start / cold start)
	bInCopyCode : BOOL;  // if TRUE, the instance afterwards gets moved into the copy code (online change)
END_VAR
eObjectType := E_BACnetObjType.ObjLoop;
END_METHOD

PROPERTY Mode : E_BACnet_LoopMode
GET
Mode := eMode;
END_GET
END_PROPERTY

PROPERTY ProportionalBand : REAL
GET
ProportionalBand := fPropBand;
END_GET
END_PROPERTY

END_FUNCTION_BLOCK

// POUs/Helper/[internal]/F_BACnet_SysTimeDiff
{attribute 'hide'} // [Workaround] Not hidden when lib is included
FUNCTION INTERNAL F_BACnet_SysTimeDiff : REAL
VAR_INPUT
	In1, In2 : T_LARGE_INTEGER;
END_VAR

F_BACnet_SysTimeDiff := LREAL_TO_REAL(INT64_TO_LREAL(Int64Sub64(In1, In2)) / 10000000.0); (* [s] *)

END_FUNCTION

// POUs/Helper/FB_BACnet_PidControl
FUNCTION_BLOCK FB_BACnet_PidControl
VAR_INPUT
	(* controller input  *)
	fSetpoint				: REAL;	(* setpoint value *)
	fPresentValue			: REAL;	(* actual value *)
	(* reset flag *)
	bReset					: BOOL;
	(* controller values *)
	fCtrlCycleTime			: REAL; (* controller cycle time in seconds [s] *)

	fBias					: REAL; (* bias also active when reset is set to 1 *)
	fKp						: REAL;	(* proportional gain Kp	(P) *)
	fKi						: REAL; (* integral gain Ki (I) *)
	fKd						: REAL;	(* derivative gain Kd (D) *)
	fTp						: REAL := -1.0;	(* damping time Tp (PT1) [s] (fTp < 0 --> Tp = Kd / 10) *)

	(* maximum ratings *)
	fMaxOutput				: REAL;
	fMinOutput				: REAL;
END_VAR
VAR_OUTPUT
	fY						: REAL; (* controller output command *)
	eErrorStatus			: E_BACnet_Error;
END_VAR
VAR
	(* Internal Variable *)
	_fE		: REAL;
	_fEOld	: REAL;
	_fYp	: REAL;
	_fYi	: REAL;
	_fYd	: REAL;
	_fbYd	: FB_BACnet_PT1;
END_VAR

(* preset error number *)
eErrorStatus	:= E_BACnet_Error.eNoError;

(* check cycle time parameter: (CycleTime > 0) *)
IF (fCtrlCycleTime <= 0.0) THEN
	eErrorStatus := E_BACnet_Error.eInvalidCycleTime;
	bReset := TRUE;
END_IF;

(* check controller parameters: (Kp, Ki, Kd >= 0) *)
IF ((fKp < 0.0) OR (fKi < 0.0) OR (fKd < 0.0)) THEN
	eErrorStatus := E_BACnet_Error.eInvalidParameter;
	bReset := TRUE;
END_IF;

(* controller reset *)
IF bReset THEN
	(* reset internal and external variables *)
	_fEOld	:= 0.0;
	fY		:= MAX(MIN(fBias, fMaxOutput), fMinOutput);
	_fYi	:= 0.0;
	_fbYd(X:= 0.0, T:= 0.0, Y=> );
	RETURN;
END_IF

(* 3. save old variable *)
_fEOld := _fE;

(* 4. set error/deviation input *)
_fE := fSetpoint - fPresentValue;

(* 5. YP-part *)
_fYp := fKp * _fE;

(* 6. YI-part *)
IF (fKi = 0.0) THEN
	_fYi	:= 0.0;
ELSE
	_fYi := _fYi + (fKi * fCtrlCycleTime * _fE);
END_IF
IF (_fYi > fMaxOutput) THEN
	(* limit wind up positive *)
	_fYi := fMaxOutput;
ELSIF (_fYi < fMinOutput) THEN
	(* limit wind up negative *)
	_fYi := fMinOutput;
END_IF

(* 7. YD-part *)
IF (fTp < 0.0) THEN
	fTp := fKd / 10.0;
END_IF
_fYd := fKd * (_fE - _fEOld) / fCtrlCycleTime;
_fbYd(X:= _fYd, T:= fTp, Tcycle:= fCtrlCycleTime, Y=> );

(* 8. Ysum = YP + YI + YD + Bias and output *)
fY := _fYp + _fYi + _fbYd.Y + fBias;
fY := MAX(MIN(fY, fMaxOutput), fMinOutput);

END_FUNCTION_BLOCK

// POUs/Helper/FB_BACnet_PT1
FUNCTION_BLOCK FB_BACnet_PT1
VAR_INPUT
	X : REAL; (* input value *)
	T : REAL; (* damping time [s] *)
	Tcycle : REAL; (* cycle time [s] of task; 0 = use internal measuring *)
END_VAR
VAR_OUTPUT
	Y : REAL; (* damped value *)
END_VAR
VAR
	_sysTime	: GETCPUCOUNTER;
	_Time		: T_LARGE_INTEGER;
	_TimeOld	: T_LARGE_INTEGER;
	_tCycleTime	: REAL;
	_Yold : REAL;
	_FirstScan : BOOL := TRUE;
END_VAR

(* determine cycle time *)
IF Tcycle = 0.0 THEN
	_TimeOld := _Time;
	_sysTime(cpuCntLoDW=> _Time.dwLowPart, cpuCntHiDW=> _Time.dwHighPart);
	_tCycleTime := F_BACnet_SysTimeDiff(In1:=_Time, In2:=_TimeOld);
ELSE
	_tCycleTime := Tcycle;
END_IF

(* exit on wrong cycle time *)
IF _tCycleTime <= 0.0 THEN
	RETURN;
END_IF

(* initialize and check on zero/negative damping time *)
IF (T <= 0.0) OR _FirstScan THEN
	Y := X;
	_Yold := Y;
	_FirstScan := FALSE;
	RETURN;
END_IF

(* remind last result *)
_Yold := Y;

(* calculate result *)
Y := 1 / ((T / _tCycleTime) + 1) * (X - _Yold) + _Yold;

END_FUNCTION_BLOCK

// POUs/Helper/FB_BACnet_AccLimit
FUNCTION_BLOCK FB_BACnet_AccLimit
VAR_INPUT
	X : REAL; (* input value [1] *)
	Amax : REAL; (* maximum acceleration of X [1/s]; 0 = limit disabled *)
	Tcycle : REAL; (* cycle time [s] of task; 0 = use internal measuring *)
END_VAR
VAR_OUTPUT
	Y : REAL; (* limited X value [1] *)
	A : REAL; (* input acceleration [1/s] *)
END_VAR
VAR
	_sysTime	: GETCPUCOUNTER;
	_Time		: T_LARGE_INTEGER;
	_TimeOld	: T_LARGE_INTEGER;
	_tCycleTime	: REAL;
	_bFirstScan	: BOOL:=TRUE;
	_foldY		: REAL;
END_VAR

(* determine cycle time *)
IF Tcycle = 0.0 THEN
	_TimeOld := _Time;
	_sysTime(cpuCntLoDW=> _Time.dwLowPart, cpuCntHiDW=> _Time.dwHighPart);
	_tCycleTime := F_BACnet_SysTimeDiff(In1:=_Time, In2:=_TimeOld);
ELSE
	_tCycleTime := Tcycle;
END_IF

IF (NOT _bFirstScan) THEN
	(* exit on wrong cycle time *)
	IF _tCycleTime <= 0.0 THEN
		RETURN;
	END_IF
	(* calculate current acceleration *)
	A := (X - _foldY) / _tCycleTime;
	IF (Amax <> 0.0) THEN
		Amax := ABS(Amax);
		IF (ABS(A) > Amax) THEN
			IF (A >= 0.0) THEN
				Y := _foldY + (Amax * _tCycleTime);
			ELSE
				Y := _foldY - (Amax * _tCycleTime);
			END_IF
		ELSE
			Y := X;
		END_IF
	ELSE
		Y := X;
	END_IF
ELSE
	Y := X;
END_IF

_foldY := Y;
_bFirstScan:=FALSE;

END_FUNCTION_BLOCK

// POUs/Local/Objects/FB_BACnet_NC
// Notification Class Object
{attribute 'enable_dynamic_creation'}
FUNCTION_BLOCK FB_BACnet_NC EXTENDS FB_BACnet_Object
VAR_INPUT CONSTANT PERSISTENT
	{region 'Variable Parameters'}
		{attribute 'parameterCategory':='Config'}
		nNotificationClass : UDINT;
		{attribute 'parameterCategory':='Config'}
		aPriority : T_BACnet_EventTransitionPriority;
		{attribute 'parameterCategory':='Config'}
		aAckRequired : T_BACnet_EventTransitions;
		{attribute 'parameterCategory':='Config'}
		aRecipientList : T_BACnet_RecipientList;
	{endregion}
END_VAR
VAR_INPUT CONSTANT
	{region 'Variable Parameters'}
		{attribute 'parameterCategory':='Config'}
		bWriteRecipientList : BOOL;
	{endregion}
END_VAR
VAR
	{region 'COV'}
		bRecipientListChanged : BOOL;
	{endregion}
END_VAR

IF (bWriteRecipientList) THEN
	// (BETA) ... [DEBUG]
	//F_BA_Print('Write RecipientList[1]', ADR(stRecipientList[1]), SIZEOF(stRecipientList[1]), TRUE, 64);
	
	bWriteRecipientList := FALSE;
	WritePropertyRecipientList(aRecipientList);
END_IF
IF (bRecipientListChanged) THEN
	bRecipientListChanged := FALSE;
	ReadPropertyRecipientList(aRecipientList);
	
	// (BETA) ... [DEBUG]
	//F_BA_Print('Read RecipientList[1]', ADR(stRecipientList[1]), SIZEOF(stRecipientList[1]), TRUE, 64);
END_IF

SUPER^();

METHOD PROTECTED OnObjectStateChanged
SUPER^.OnObjectStateChanged();

CASE (tState) OF
	TCOM_STATE.TCOM_STATE_PREOP:
		// SyncHandler:
		RequestSyncHandlers(0, 7);
		
	TCOM_STATE.TCOM_STATE_SAFEOP:
		;
		
	TCOM_STATE.TCOM_STATE_OP:
		IF (SyncPropertyCOV(E_BACnetPropIdentifier.PropRecipientList, ADR(bRecipientListChanged))) THEN
			WritePropertyRecipientList(aRecipientList);
		END_IF
		
		SyncProperty(E_BACnetPropIdentifier.PropNotificationClass, SIZEOF(nNotificationClass), ADR(nNotificationClass), 0, eFullSync_InitPLC, FALSE);
		SyncPropertyIdx(E_BACnetPropIdentifier.PropPriority, SIZEOF(UDINT), ADR(aPriority[E_BA_EventTransition.eToOffnormal]), (E_BACnet_EventTransitionBits.eToOffnormal+1), 0, eFullSync_InitPLC, FALSE);	
		SyncPropertyIdx(E_BACnetPropIdentifier.PropPriority, SIZEOF(UDINT), ADR(aPriority[E_BA_EventTransition.eToFault]), (E_BACnet_EventTransitionBits.eToFault+1), 0, eFullSync_InitPLC, FALSE);	
		SyncPropertyIdx(E_BACnetPropIdentifier.PropPriority, SIZEOF(UDINT), ADR(aPriority[E_BA_EventTransition.eToNormal]), (E_BACnet_EventTransitionBits.eToNormal+1), 0, eFullSync_InitPLC, FALSE);
		SyncPropertyIdx(E_BACnetPropIdentifier.PropAckRequired, SIZEOF(BOOL), ADR(aAckRequired[E_BA_EventTransition.eToOffnormal]), E_BACnet_EventTransitionBits.eToOffnormal, 0, eFullSync_InitPLC, FALSE);	
		SyncPropertyIdx(E_BACnetPropIdentifier.PropAckRequired, SIZEOF(BOOL), ADR(aAckRequired[E_BA_EventTransition.eToFault]), E_BACnet_EventTransitionBits.eToFault, 0, eFullSync_InitPLC, FALSE);	
		SyncPropertyIdx(E_BACnetPropIdentifier.PropAckRequired, SIZEOF(BOOL), ADR(aAckRequired[E_BA_EventTransition.eToNormal]), E_BACnet_EventTransitionBits.eToNormal, 0, eFullSync_InitPLC, FALSE);
		
END_CASE
END_METHOD

METHOD FB_init : BOOL
VAR_INPUT
	bInitRetains : BOOL; // if TRUE, the retain variables are initialized (warm start / cold start)
	bInCopyCode : BOOL;  // if TRUE, the instance afterwards gets moved into the copy code (online change)
END_VAR
eObjectType := E_BACnetObjType.ObjNotificationClass;
END_METHOD

END_FUNCTION_BLOCK

// POUs/Local/Objects/FB_BACnet_Prog
// Program Object
{attribute 'enable_dynamic_creation'}
FUNCTION_BLOCK FB_BACnet_Prog EXTENDS FB_BACnet_Object
VAR_OUTPUT
	eState			: E_BACnet_ProgramState;
END_VAR

SUPER^();

METHOD PROTECTED OnObjectStateChanged
SUPER^.OnObjectStateChanged();

CASE (tState) OF
	TCOM_STATE.TCOM_STATE_PREOP:
		// SyncHandler:
		RequestSyncHandlers(1, 0);
		
	TCOM_STATE.TCOM_STATE_SAFEOP:
		;
	
	TCOM_STATE.TCOM_STATE_OP:
		SyncProperty(E_BACnetPropIdentifier.PropProgramState, SIZEOF(eState), ADR(eState), 0, eSync_FromSupplement, FALSE);
		
END_CASE
END_METHOD

METHOD FB_init : BOOL
VAR_INPUT
	bInitRetains : BOOL; // if TRUE, the retain variables are initialized (warm start / cold start)
	bInCopyCode : BOOL;  // if TRUE, the instance afterwards gets moved into the copy code (online change)
END_VAR
eObjectType := E_BACnetObjType.ObjProg;
END_METHOD

END_FUNCTION_BLOCK

// POUs/Local/Objects/FB_BACnet_SchedA
// Analog Scheduler Object
{attribute 'enable_dynamic_creation'}
FUNCTION_BLOCK FB_BACnet_SchedA EXTENDS FB_BACnet_BaseSched
VAR_INPUT CONSTANT PERSISTENT
	{region 'Fixed Parameters'}
		{attribute 'parameterCategory':='Value'}
		fScheduleDefault : REAL;
	{endregion}
END_VAR
VAR_OUTPUT
	fPresentValue		: REAL;
END_VAR

SUPER^();

METHOD PROTECTED OnObjectStateChanged
SUPER^.OnObjectStateChanged();

CASE (tState) OF
	TCOM_STATE.TCOM_STATE_PREOP:
		// SyncHandler:
		RequestSyncHandlers(1, 6);
		
	TCOM_STATE.TCOM_STATE_SAFEOP:
		;
		
	TCOM_STATE.TCOM_STATE_OP:
		SyncProperty(E_BACnetPropIdentifier.PropPresentValueReal, SIZEOF(fPresentValue), ADR(fPresentValue), 0, eSync_FromSupplement, FALSE);	
		WritePropertyValueEx(E_BACnetPropIdentifier.PropScheduleDefault, eDatatype, SIZEOF(fScheduleDefault), ADR(fScheduleDefault));
END_CASE
END_METHOD

METHOD FB_init : BOOL
VAR_INPUT
	bInitRetains : BOOL; // if TRUE, the retain variables are initialized (warm start / cold start)
	bInCopyCode : BOOL;  // if TRUE, the instance afterwards gets moved into the copy code (online change)
END_VAR
eDatatype := E_BACnet_ValueChoice.eRealValue;

// Init default values:
aWeek := F_BACnet_SchedWeekly1xA(E_BA_Weekday.eMonday, E_BA_Weekday.eFriday, T#0H, 0.0);
END_METHOD

END_FUNCTION_BLOCK

// POUs/Local/Objects/[Base]/FB_BACnet_BaseSched
FUNCTION_BLOCK FB_BACnet_BaseSched EXTENDS FB_BACnet_Object
VAR_INPUT CONSTANT PERSISTENT
	{region 'Variable Parameters'}
		{attribute 'parameterCategory':='Value'}
		aWeek : T_BACnet_SchedWeek;															// Entries (separated per days) for weekly organization
		{attribute 'parameterCategory':='Value'}
		aCalendar : T_BACnet_SchedCalendar;													// Entries (separated per calendar) for global (calendar) exceptions organization (See "fbCalendar")
		{attribute 'parameterCategory':='Value'}
		aException : T_BACnet_SchedExceptionList;											// Entries (separated per exception count) for local (Presrent instance) exceptions organization
			 
		{attribute 'parameterCategory':='Config'}
		stObjectPropertyReference : ST_BACnet_ObjectPropertyReference;
	{endregion}
END_VAR
VAR_INPUT CONSTANT
	{region 'Variable Parameters'}
		{attribute 'parameterCategory':='Value'}
		bWriteWeekly : BOOL;
		{attribute 'parameterCategory':='Value'}
		bWriteException : BOOL;
	{endregion}
END_VAR
VAR	
	{region 'COV'}
		bWeeklyChanged			: BOOL;
		bExceptionChanged		: BOOL;
	{endregion}
END_VAR
VAR
	{region 'Internal'}
		eDatatype				: E_BACnet_ValueChoice					:= E_BACnet_ValueChoice.eNullValue;
	{endregion}
END_VAR

IF (bWriteWeekly OR bWriteException) THEN
	WriteContent(bWriteWeekly, bWriteException);
	
	bWriteWeekly := FALSE;
	bWriteException := FALSE;
END_IF
IF (bWeeklyChanged OR bExceptionChanged) THEN
	ReadContent(bWeeklyChanged, bExceptionChanged);
	
	bWeeklyChanged := FALSE;
	bExceptionChanged := FALSE;
END_IF

SUPER^();

METHOD PROTECTED OnObjectStateChanged
SUPER^.OnObjectStateChanged();

CASE (tState) OF
	TCOM_STATE.TCOM_STATE_PREOP:
		// SyncHandler:
		RequestSyncHandlers(2, 0);
		
		// Properties:
		WriteProtectProperty(E_BACnetPropIdentifier.PropScheduleDefault, TRUE);
	
	TCOM_STATE.TCOM_STATE_SAFEOP:
		;
		
	TCOM_STATE.TCOM_STATE_OP:
		// Validate referred property:
		IF (ValidateReference(stObjectPropertyReference.iObject, stObjectPropertyReference.tObjectID, 16#FF)) THEN
			ObjectPropertyReference := stObjectPropertyReference;
		END_IF
		
		SyncPropertyCOV(E_BACnetPropIdentifier.PropWeeklySchedule, ADR(bWeeklyChanged));
		SyncPropertyCOV(E_BACnetPropIdentifier.PropExceptionSchedule, ADR(bExceptionChanged));
	
		WriteContent(TRUE, TRUE);
		WritePropertyUDInt(E_BACnetPropIdentifier.PropPriorityForWriting, BACnet_Param.nSched_PrioForWriting);
		
END_CASE
END_METHOD

METHOD FB_init : BOOL
VAR_INPUT
	bInitRetains : BOOL; // if TRUE, the retain variables are initialized (warm start / cold start)
	bInCopyCode : BOOL;  // if TRUE, the instance afterwards gets moved into the copy code (online change)
END_VAR
eObjectType := E_BACnetObjType.ObjSchedule;
END_METHOD

METHOD ReadContent : BOOL
VAR_INPUT
	bWeeklySched		: BOOL		:= TRUE;
	bExceptSched		: BOOL		:= TRUE;
END_VAR
IF (bWeeklySched) THEN
	IF (ReadPropertyWeeklySched(aWeek, eDataType) <> S_OK) THEN
		RETURN;
	END_IF
END_IF
IF (bExceptSched) THEN
	IF (ReadPropertyExceptionSched(aCalendar, aException, eDataType) <> S_OK) THEN
		RETURN;
	END_IF
END_IF

ReadContent := TRUE;
END_METHOD

METHOD WriteContent : BOOL
VAR_INPUT
	bWeeklySched		: BOOL		:= TRUE;
	bExceptSched		: BOOL		:= TRUE;
END_VAR
WriteContent := TRUE;

IF (bWeeklySched) THEN
	_hResult := WritePropertyWeeklySched(aWeek, eDataType);
	WriteContent := (WriteContent) AND (_hResult=S_OK);
	bWeeklyChanged := FALSE;
END_IF
IF (bExceptSched) THEN
	_hResult := WritePropertyExceptionSched(aCalendar, aException, eDataType);
	WriteContent := (WriteContent) AND (_hResult=S_OK);
	bExceptionChanged := FALSE;
END_IF
END_METHOD

PROPERTY ObjectPropertyReference : ST_BACnet_ObjectPropertyReference
GET
ObjectPropertyReference := stObjectPropertyReference;
END_GET
SET
stObjectPropertyReference := ObjectPropertyReference;

WritePropertyReferenceList1x(E_BACnetPropIdentifier.PropListOfObjectPropertyReferences, stObjectPropertyReference);
END_SET
END_PROPERTY

END_FUNCTION_BLOCK

// POUs/Helper/Scheduler/Weekly/F_BACnet_SchedWeekly1xA
// Returns an initialized analog weekly scheduler.
FUNCTION F_BACnet_SchedWeekly1xA : T_BACnet_SchedWeek
VAR_INPUT
	eDayFrom		: E_BA_Weekday		:= E_BA_Weekday.eMonday;
	eDayTo			: E_BA_Weekday		:= E_BA_Weekday.eSunday;
	
	tEntry1Time		: TIME;
	fEntry1Value	: REAL;
END_VAR

F_BA_SetWeekdays(F_BACnet_SchedWeekly1xA, eDayFrom, eDayTo, 1, tEntry1Time, F_BA_RVal(fEntry1Value));

END_FUNCTION

// POUs/Local/Objects/FB_BACnet_SchedB
// Binary Scheduler Object
{attribute 'enable_dynamic_creation'}
FUNCTION_BLOCK FB_BACnet_SchedB EXTENDS FB_BACnet_BaseSched
VAR_INPUT
	{attribute 'parameterUnit':= 's'}
	nPredictTime : UDINT;
END_VAR
VAR_INPUT CONSTANT PERSISTENT
	{region 'Fixed Parameters'}
		{attribute 'parameterCategory':='Value'}
		bScheduleDefault 	: BOOL;
	{endregion}
END_VAR
VAR_OUTPUT
	bPresentValue			: BOOL;
	bPredictedValue			: BOOL;
END_VAR

SUPER^();

METHOD PROTECTED OnObjectStateChanged
VAR
	_ePropPresentVal		: E_BACnetPropIdentifier;
END_VAR
SUPER^.OnObjectStateChanged();

CASE (tState) OF
	TCOM_STATE.TCOM_STATE_PREOP:
		// SyncHandler:
		RequestSyncHandlers(2, 1);
		
	TCOM_STATE.TCOM_STATE_SAFEOP:
		;
		
	TCOM_STATE.TCOM_STATE_OP:
		CASE (eDatatype) OF
			E_BACnet_ValueChoice.eEnumerationValue:
				_ePropPresentVal := E_BACnetPropIdentifier.PropPresentValueEnumerated;
			E_BACnet_ValueChoice.eBoolValue:
				_ePropPresentVal := E_BACnetPropIdentifier.PropPresentValueBool;
		ELSE
			iOwner.LogMsg.Show1(ADSLOG_MSGTYPE_ERROR, 'OOSC17', 'Property-synchronization aborted: Invalid datatype "%d"!', F_INT(eDatatype), FALSE);		
			RETURN;
		END_CASE

		SyncProperty(_ePropPresentVal, SIZEOF(bPresentValue), ADR(bPresentValue), 0, eSync_FromSupplement, FALSE);
		SyncProperty(E_BACnetPropIdentifier.PropPredictedScheduleBoolValue, SIZEOF(bPredictedValue), ADR(bPredictedValue), 0, eSync_FromSupplement, FALSE);

		SyncProperty(E_BACnetPropIdentifier.PropPredictScheduleValueTime, SIZEOF(nPredictTime), ADR(nPredictTime), 0, eSync_ToSupplement, FALSE);

		WritePropertyValueEx(E_BACnetPropIdentifier.PropScheduleDefault, eDatatype, SIZEOF(bScheduleDefault), ADR(bScheduleDefault));
		
END_CASE
END_METHOD

METHOD FB_init : BOOL
VAR_INPUT
	bInitRetains : BOOL; // if TRUE, the retain variables are initialized (warm start / cold start)
	bInCopyCode : BOOL;  // if TRUE, the instance afterwards gets moved into the copy code (online change)
END_VAR
CASE (BACnet_Param.eSched_BType) OF
	E_BACnet_SchedBType.eBinaryPV:
		eDatatype := E_BACnet_ValueChoice.eEnumerationValue;
	E_BACnet_SchedBType.eBool:
		eDatatype := E_BACnet_ValueChoice.eBoolValue;
END_CASE

// Init default values:
aWeek := F_BACnet_SchedWeekly1xB(E_BA_Weekday.eMonday, E_BA_Weekday.eFriday, T#0H, FALSE);
END_METHOD

END_FUNCTION_BLOCK

// POUs/Helper/Scheduler/Weekly/F_BACnet_SchedWeekly1xB
// Returns an initialized binary weekly scheduler.
FUNCTION F_BACnet_SchedWeekly1xB : T_BACnet_SchedWeek
VAR_INPUT
	eDayFrom		: E_BA_Weekday		:= E_BA_Weekday.eMonday;
	eDayTo			: E_BA_Weekday		:= E_BA_Weekday.eSunday;
	
	tEntry1Time		: TIME;
	bEntry1Value	: BOOL;
END_VAR

F_BA_SetWeekdays(F_BACnet_SchedWeekly1xB, eDayFrom, eDayTo, 1, tEntry1Time, F_BA_BVal(bEntry1Value));

END_FUNCTION

// POUs/Local/Objects/FB_BACnet_SchedM
// Multistate Scheduler Object
{attribute 'enable_dynamic_creation'}
FUNCTION_BLOCK FB_BACnet_SchedM EXTENDS FB_BACnet_BaseSched
VAR_INPUT CONSTANT PERSISTENT
	{region 'Fixed Parameters'}
		{attribute 'parameterCategory':='Value'}
		nScheduleDefault : UDINT;
	{endregion}
END_VAR
VAR_OUTPUT
	nPresentValue		: UDINT;
END_VAR

SUPER^();

METHOD PROTECTED OnObjectStateChanged
SUPER^.OnObjectStateChanged();

CASE (tState) OF
	TCOM_STATE.TCOM_STATE_PREOP:
		// SyncHandler:
		RequestSyncHandlers(1, 0);
		
	TCOM_STATE.TCOM_STATE_SAFEOP:
		;
		
	TCOM_STATE.TCOM_STATE_OP:
		SyncProperty(E_BACnetPropIdentifier.PropPresentValueUnsigned, SIZEOF(nPresentValue), ADR(nPresentValue), 0, eSync_FromSupplement, FALSE);
		
		WritePropertyValueEx(E_BACnetPropIdentifier.PropScheduleDefault, eDatatype, SIZEOF(nScheduleDefault), ADR(nScheduleDefault));
		
END_CASE
END_METHOD

METHOD FB_init : BOOL
VAR_INPUT
	bInitRetains : BOOL; // if TRUE, the retain variables are initialized (warm start / cold start)
	bInCopyCode : BOOL;  // if TRUE, the instance afterwards gets moved into the copy code (online change)
END_VAR
eDatatype := E_BACnet_ValueChoice.eUnsignedValue;

// Init default values:
aWeek := F_BACnet_SchedWeekly1xM(E_BA_Weekday.eMonday, E_BA_Weekday.eFriday, T#0H, 1);
END_METHOD

END_FUNCTION_BLOCK

// POUs/Helper/Scheduler/Weekly/F_BACnet_SchedWeekly1xM
// Returns an initialized multistate weekly scheduler.
FUNCTION F_BACnet_SchedWeekly1xM : T_BACnet_SchedWeek
VAR_INPUT
	eDayFrom		: E_BA_Weekday		:= E_BA_Weekday.eMonday;
	eDayTo			: E_BA_Weekday		:= E_BA_Weekday.eSunday;
	
	tEntry1Time		: TIME;
	nEntry1Value	: UDINT;
END_VAR

F_BA_SetWeekdays(F_BACnet_SchedWeekly1xM, eDayFrom, eDayTo, 1, tEntry1Time, F_BA_UDIVal(nEntry1Value));

END_FUNCTION

// POUs/Local/Objects/FB_BACnet_Acc
// Accumulator Object
{attribute 'enable_dynamic_creation'}
FUNCTION_BLOCK FB_BACnet_Acc EXTENDS FB_BACnet_EventObject
VAR_OUTPUT
	nPresentValue			: UDINT;
END_VAR

SUPER^();

METHOD PROTECTED OnObjectStateChanged
SUPER^.OnObjectStateChanged();

CASE (tState) OF
	TCOM_STATE.TCOM_STATE_PREOP:
		// SyncHandler:
		RequestSyncHandlers(1, 0);
		
	TCOM_STATE.TCOM_STATE_SAFEOP:
		SyncProperty(E_BACnetPropIdentifier.PropPresentValue, SIZEOF(nPresentValue), ADR(nPresentValue), 0, eSync_FromSupplement, TRUE);
	
	TCOM_STATE.TCOM_STATE_OP:
		;
		
END_CASE
END_METHOD

METHOD FB_init : BOOL
VAR_INPUT
	bInitRetains : BOOL; // if TRUE, the retain variables are initialized (warm start / cold start)
	bInCopyCode : BOOL;  // if TRUE, the instance afterwards gets moved into the copy code (online change)
END_VAR
eObjectType := E_BACnetObjType.ObjAccumulator;
END_METHOD

END_FUNCTION_BLOCK

// POUs/Local/Objects/FB_BACnet_PC
// Pulse Converter Object
{attribute 'enable_dynamic_creation'}
FUNCTION_BLOCK FB_BACnet_PC EXTENDS FB_BACnet_EventObject
VAR_OUTPUT
	fPresentValue			: REAL;
END_VAR

SUPER^();

METHOD PROTECTED OnObjectStateChanged
SUPER^.OnObjectStateChanged();

CASE (tState) OF
	TCOM_STATE.TCOM_STATE_PREOP:
		// SyncHandler:
		RequestSyncHandlers(1, 0);
		
	TCOM_STATE.TCOM_STATE_SAFEOP:
		SyncProperty(E_BACnetPropIdentifier.PropPresentValue, SIZEOF(fPresentValue), ADR(fPresentValue), 0, eSync_FromSupplement, TRUE);
	
	TCOM_STATE.TCOM_STATE_OP:
		;
		
END_CASE
END_METHOD

METHOD FB_init : BOOL
VAR_INPUT
	bInitRetains : BOOL; // if TRUE, the retain variables are initialized (warm start / cold start)
	bInCopyCode : BOOL;  // if TRUE, the instance afterwards gets moved into the copy code (online change)
END_VAR
eObjectType := E_BACnetObjType.ObjPulseConverter;
END_METHOD

END_FUNCTION_BLOCK

// POUs/Helper/[internal]/Calendar/F_BACnet_CopyDateListEntry
{attribute 'hide'} // [Workaround] Not hidden when lib is included
FUNCTION INTERNAL F_BACnet_ToDateListEntry : BOOL
VAR_INPUT
	stEntry		: POINTER TO ST_BA_CalendarEntry;
END_VAR
VAR_OUTPUT
	stResult	: ST_BACnet_CalendarEntry;
END_VAR

IF (stEntry <> 0) AND_THEN (F_BA_IsDateValChoiceValid(stEntry^.eType)) THEN
	// Clear contents:
	MEMSET(ADR(stResult), 0, SIZEOF(ST_BACnet_CalendarEntry));
 
	CASE (stEntry^.eType) OF
		E_BA_DateValChoice.eDate:
			stResult.uCalEntry.stDate := stEntry^.uDate.stDate;
		E_BA_DateValChoice.eDateRange:
			stResult.uCalEntry.stDateRange := stEntry^.uDate.stDateRange;
		E_BA_DateValChoice.eWeekNDay:
			stResult.uCalEntry.stWeekNDay := stEntry^.uDate.stWeekNDay;
	ELSE
		RETURN;
	END_CASE
	
	stResult.eEventChoice := (stEntry^.eType-1);
	
	F_BACnet_ToDateListEntry := TRUE;
END_IF

END_FUNCTION

// POUs/Helper/[internal]/Remote/F_BACnetRM_GetWriteEntrySize
FUNCTION F_BACnetRM_GetWriteEntrySize : UDINT
VAR_INPUT
	entry : ST_BACnetRM_WriteEntry;
END_VAR
VAR
END_VAR

IF entry.pNull <> 0 AND_THEN entry.pNull^ THEN
	F_BACnetRM_GetWriteEntrySize:=0;
	RETURN;
END_IF
IF entry.ePropID = E_BACnetPropIdentifier.PropEventEnable OR  entry.ePropID = E_BACnetPropIdentifier.PropLimitEnable THEN
	F_BACnetRM_GetWriteEntrySize:=2;
	RETURN;
END_IF

F_BACnetRM_GetWriteEntrySize:=entry.nData;

END_FUNCTION

// POUs/Helper/[internal]/Remote/F_BACnetRM_IsErrorSet
{attribute 'hide'}
FUNCTION F_BACnetRM_IsErrorSet : BOOL
VAR_INPUT
	stResult	: POINTER TO SendDataRequestResult;
END_VAR
VAR
END_VAR

F_BACnetRM_IsErrorSet:=TRUE;
IF stResult^.errorType = E_BACnet_ErrorType.eAbort AND stResult^.abortReason = E_BACnet_AbortReason.NoReason THEN
	F_BACnetRM_IsErrorSet:=FALSE;
	RETURN;
END_IF
IF stResult^.errorType = E_BACnet_ErrorType.eError AND stResult^.errorClass = E_BACnet_ErrorClass.NoError THEN
	F_BACnetRM_IsErrorSet:=FALSE;
	RETURN;
END_IF
IF stResult^.errorType = E_BACnet_ErrorType.eReject AND stResult^.rejectCode = E_BACnet_RejectReason.NoReason THEN
	F_BACnetRM_IsErrorSet:=FALSE;
	RETURN;
END_IF

END_FUNCTION

// POUs/Helper/[internal]/Remote/F_IsCovProperty
FUNCTION F_IsCovProperty : BOOL
VAR_INPUT
	eObjectType			: E_BACnetObjType;
	ePropID				: E_BACnetPropIdentifier;
END_VAR

CASE eObjectType OF
	E_BACnetObjType.ObjAnalogInput:
		IF ePropID = E_BACnetPropIdentifier.PropPresentValue OR ePropID = E_BACnetPropIdentifier.PropStatusFlags THEN
			F_IsCovProperty:=TRUE;
		END_IF
	E_BACnetObjType.ObjAnalogOutput:
		IF ePropID = E_BACnetPropIdentifier.PropPresentValue OR ePropID = E_BACnetPropIdentifier.PropStatusFlags THEN
			F_IsCovProperty:=TRUE;
		END_IF
	E_BACnetObjType.ObjAnalogValue:
		IF ePropID = E_BACnetPropIdentifier.PropPresentValue OR ePropID = E_BACnetPropIdentifier.PropStatusFlags THEN
			F_IsCovProperty:=TRUE;
		END_IF
	E_BACnetObjType.ObjBinaryInput:
		IF ePropID = E_BACnetPropIdentifier.PropPresentValue OR ePropID = E_BACnetPropIdentifier.PropStatusFlags THEN
			F_IsCovProperty:=TRUE;
		END_IF
	E_BACnetObjType.ObjBinaryOutput:
		IF ePropID = E_BACnetPropIdentifier.PropPresentValue OR ePropID = E_BACnetPropIdentifier.PropStatusFlags THEN
			F_IsCovProperty:=TRUE;
		END_IF
	E_BACnetObjType.ObjBinaryValue:
		IF ePropID = E_BACnetPropIdentifier.PropPresentValue OR ePropID = E_BACnetPropIdentifier.PropStatusFlags THEN
			F_IsCovProperty:=TRUE;
		END_IF
	E_BACnetObjType.ObjMultiStateInput:
		IF ePropID = E_BACnetPropIdentifier.PropPresentValue OR ePropID = E_BACnetPropIdentifier.PropStatusFlags THEN
			F_IsCovProperty:=TRUE;
		END_IF
	E_BACnetObjType.ObjMultiStateOutput:
		IF ePropID = E_BACnetPropIdentifier.PropPresentValue OR ePropID = E_BACnetPropIdentifier.PropStatusFlags THEN
			F_IsCovProperty:=TRUE;
		END_IF
	E_BACnetObjType.ObjMultiStateValue:
		IF ePropID = E_BACnetPropIdentifier.PropPresentValue OR ePropID = E_BACnetPropIdentifier.PropStatusFlags THEN
			F_IsCovProperty:=TRUE;
		END_IF
	E_BACnetObjType.ObjLargeAnalogValue:
		IF ePropID = E_BACnetPropIdentifier.PropPresentValue OR ePropID = E_BACnetPropIdentifier.PropStatusFlags THEN
			F_IsCovProperty:=TRUE;
		END_IF
	E_BACnetObjType.ObjPositiveIntegerValue:
		IF ePropID = E_BACnetPropIdentifier.PropPresentValue OR ePropID = E_BACnetPropIdentifier.PropStatusFlags THEN
			F_IsCovProperty:=TRUE;
		END_IF
	E_BACnetObjType.ObjIntegerValue:
		IF ePropID = E_BACnetPropIdentifier.PropPresentValue OR ePropID = E_BACnetPropIdentifier.PropStatusFlags THEN
			F_IsCovProperty:=TRUE;
		END_IF
	E_BACnetObjType.ObjOctetStringValue:
		IF ePropID = E_BACnetPropIdentifier.PropPresentValue OR ePropID = E_BACnetPropIdentifier.PropStatusFlags THEN
			F_IsCovProperty:=TRUE;
		END_IF
	E_BACnetObjType.ObjCharacterStringValue:
		IF ePropID = E_BACnetPropIdentifier.PropPresentValue OR ePropID = E_BACnetPropIdentifier.PropStatusFlags THEN
			F_IsCovProperty:=TRUE;
		END_IF
	E_BACnetObjType.ObjTimePatternValue:
		IF ePropID = E_BACnetPropIdentifier.PropPresentValue OR ePropID = E_BACnetPropIdentifier.PropStatusFlags THEN
			F_IsCovProperty:=TRUE;
		END_IF
	E_BACnetObjType.ObjTimeValue:
		IF ePropID = E_BACnetPropIdentifier.PropPresentValue OR ePropID = E_BACnetPropIdentifier.PropStatusFlags THEN
			F_IsCovProperty:=TRUE;
		END_IF
	E_BACnetObjType.ObjDatePatternValue:
		IF ePropID = E_BACnetPropIdentifier.PropPresentValue OR ePropID = E_BACnetPropIdentifier.PropStatusFlags THEN
			F_IsCovProperty:=TRUE;
		END_IF
	E_BACnetObjType.ObjDateValue:
		IF ePropID = E_BACnetPropIdentifier.PropPresentValue OR ePropID = E_BACnetPropIdentifier.PropStatusFlags THEN
			F_IsCovProperty:=TRUE;
		END_IF
	E_BACnetObjType.ObjDateTimePatternValue:
		IF ePropID = E_BACnetPropIdentifier.PropPresentValue OR ePropID = E_BACnetPropIdentifier.PropStatusFlags THEN
			F_IsCovProperty:=TRUE;
		END_IF
	E_BACnetObjType.ObjDateTimeValue:
		IF ePropID = E_BACnetPropIdentifier.PropPresentValue OR ePropID = E_BACnetPropIdentifier.PropStatusFlags THEN
			F_IsCovProperty:=TRUE;
		END_IF
	E_BACnetObjType.ObjLoop:
		IF ePropID = E_BACnetPropIdentifier.PropPresentValue OR ePropID = E_BACnetPropIdentifier.PropStatusFlags OR ePropID = E_BACnetPropIdentifier.PropSetpoint OR ePropID = E_BACnetPropIdentifier.PropControlledVariableValue THEN
			F_IsCovProperty:=TRUE;
		END_IF
	E_BACnetObjType.ObjPulseConverter:
			IF ePropID = E_BACnetPropIdentifier.PropPresentValue OR ePropID = E_BACnetPropIdentifier.PropStatusFlags OR ePropID = E_BACnetPropIdentifier.PropUpdateTime THEN
			F_IsCovProperty:=TRUE;
		END_IF
END_CASE

END_FUNCTION

// POUs/Helper/[internal]/Remote/F_IsCovReadMode
FUNCTION F_IsCovReadMode : BOOL
VAR_INPUT
	eReadMode : E_BACnet_CommMode;
END_VAR

IF eReadMode = E_BACnet_CommMode.eCov OR eReadMode = E_BACnet_CommMode.eCovC OR eReadMode = E_BACnet_CommMode.eCovU THEN
	F_IsCovReadMode:=TRUE;
END_IF

END_FUNCTION

// POUs/Helper/[internal]/Remote/F_IsCovReqType
FUNCTION F_IsCovReqType : BOOL
VAR_INPUT
	iReq : I_BACnetRM_BaseReq;
END_VAR
VAR
	tmpReqType : E_BACnetRM_RequestType;
END_VAR

tmpReqType := iReq.GetRequestType();

IF tmpReqType = E_BACnetRM_RequestType.eCOV OR tmpReqType = E_BACnetRM_RequestType.eCOV_C OR tmpReqType = E_BACnetRM_RequestType.eCOV_U THEN
	F_IsCovReqType:=TRUE;
END_IF

END_FUNCTION

// POUs/Helper/[internal]/Validation-Functions/F_BACnet_IsAbortReasonValid
{attribute 'hide'} // [Workaround] Not hidden when lib is included
FUNCTION INTERNAL F_BACnet_IsAbortReasonValid : BOOL
VAR_INPUT
	eReason		: E_BACnet_AbortReason;
END_VAR

F_BACnet_IsAbortReasonValid := (E_BACnet_AbortReason.First <= eReason) AND_THEN (eReason <= E_BACnet_AbortReason.Last);

END_FUNCTION

// POUs/Helper/[internal]/Validation-Functions/F_BACnet_IsErrorClassValid
{attribute 'hide'} // [Workaround] Not hidden when lib is included
FUNCTION INTERNAL F_BACnet_IsErrorClassValid : BOOL
VAR_INPUT
	eClass		: E_BACnet_ErrorClass;
END_VAR

F_BACnet_IsErrorClassValid := (E_BACnet_ErrorClass.First <= eClass) AND_THEN (eClass <= E_BACnet_ErrorClass.Last);

END_FUNCTION

// POUs/Helper/[internal]/Validation-Functions/F_BACnet_IsErrorCodeValid
{attribute 'hide'} // [Workaround] Not hidden when lib is included
FUNCTION INTERNAL F_BACnet_IsErrorCodeValid : BOOL
VAR_INPUT
	eCode		: E_BACnet_ErrorCode;
END_VAR

F_BACnet_IsErrorCodeValid := (E_BACnet_ErrorCode.First <= eCode) AND_THEN (eCode <= E_BACnet_ErrorCode.Last);

END_FUNCTION

// POUs/Helper/[internal]/Validation-Functions/F_BACnet_IsErrorTypeValid
{attribute 'hide'} // [Workaround] Not hidden when lib is included
FUNCTION INTERNAL F_BACnet_IsErrorTypeValid : BOOL
VAR_INPUT
	eType		: E_BACnet_ErrorType;
END_VAR

F_BACnet_IsErrorTypeValid := (E_BACnet_ErrorType.First <= eType) AND_THEN (eType <= E_BACnet_ErrorType.Last);

END_FUNCTION

// POUs/Helper/[internal]/Validation-Functions/F_BACnet_IsPropIdentifierValid
{attribute 'hide'} // [Workaround] Not hidden when lib is included
FUNCTION INTERNAL F_BACnet_IsPropIdentifierValid : BOOL
VAR_INPUT
	eProperty		: E_BACnetPropIdentifier;
END_VAR

F_BACnet_IsPropIdentifierValid := (eProperty <> E_BACnetPropIdentifier.PropInvalid);

END_FUNCTION

// POUs/Helper/[internal]/Validation-Functions/F_BACnet_IsRejectReasonValid
{attribute 'hide'} // [Workaround] Not hidden when lib is included
FUNCTION INTERNAL F_BACnet_IsRejectReasonValid : BOOL
VAR_INPUT
	eReason		: E_BACnet_RejectReason;
END_VAR

F_BACnet_IsRejectReasonValid := (E_BACnet_RejectReason.First <= eReason) AND_THEN (eReason <= E_BACnet_RejectReason.Last);

END_FUNCTION

// POUs/Helper/[internal]/F_BACnet_AnalogPV
{attribute 'hide'} // [Workaround] Not hidden when lib is included
FUNCTION INTERNAL F_BACnet_AnalogPV : REAL
VAR_INPUT
	bEnable	: BOOL; (* TRUE = commit to stack, FALSE = do-nothing *)
	bNull	: BOOL; (* TRUE = clear priority, FALSE = write value from input *)
	fValue	: REAL;
END_VAR
VAR
	pres : POINTER TO DWORD;
END_VAR

IF (bEnable) THEN
	IF (bNull) THEN
		pres := ADR(F_BACnet_AnalogPV);
		pres^ := F_BACnet_RealNull(); 
	ELSE
		F_BACnet_AnalogPV := fValue;
	END_IF
ELSE
	F_BACnet_AnalogPV := F_BACnet_NAN();
END_IF

END_FUNCTION

// POUs/Helper/Real/F_BACnet_RealNull
FUNCTION F_BACnet_RealNull : DWORD
(* function that generates <not-a-number> real state *)

F_BACnet_RealNull:=16#7FFF0000;

END_FUNCTION

// POUs/Helper/Real/F_BACnet_NAN
FUNCTION F_BACnet_NAN : REAL
(* function that generates <not-a-number> real state *)
VAR
	res : POINTER TO DWORD;
END_VAR

res:=ADR(F_BACnet_NAN);
res^:=16#7FFFFFFF;

END_FUNCTION

// POUs/Helper/[internal]/F_BACnet_ChangeBitFieldBit
{attribute 'hide'} // [Workaround] Not hidden when lib is included
FUNCTION INTERNAL F_BACnet_ChangeBitFieldBit : DWORD
VAR_INPUT
	ptrData		: POINTER TO DWORD;
	bitNbr			: INT;
	Value		: BOOL;
END_VAR
VAR
END_VAR

IF (NOT Value) THEN
	ptrData^ := ptrData^ AND NOT (SHR(DWORD#16#00008000,F_BACnet_BitFieldBit(bitNbr)));
ELSE
	ptrData^ := ptrData^ OR (SHR(DWORD#16#00008000,F_BACnet_BitFieldBit(bitNbr)));
END_IF
F_BACnet_ChangeBitFieldBit := ptrData^;

END_FUNCTION

// POUs/Helper/[internal]/F_BACnet_ElemSize
FUNCTION F_BACnet_ElemSize : UDINT
VAR_INPUT
	nSize : UDINT;
END_VAR

F_BACnet_ElemSize := (nSize AND 16#7FFFFFFF);

END_FUNCTION

// POUs/Helper/[internal]/F_BACnet_IsBitFieldBitSetPtr
{attribute 'hide'} // [Workaround] Not hidden when lib is included
FUNCTION INTERNAL F_BACnet_IsBitFieldBitSetPtr : BOOL
VAR_INPUT
	pData	:	POINTER TO WORD;
	bitNbr	:	INT;
END_VAR
VAR
END_VAR

F_BACnet_IsBitFieldBitSetPtr:= ((pData^) AND (SHR(16#8000,F_BACnet_BitFieldBit(bitNbr)))) > 0;

END_FUNCTION

// POUs/Helper/[internal]/F_BACnet_UnSetBitFieldBit
{attribute 'hide'} // [Workaround] Not hidden when lib is included
FUNCTION INTERNAL F_BACnet_UnSetBitFieldBit : DWORD
VAR_INPUT
	ptrData		:	POINTER TO DWORD;
	bitNbr			:	INT;
END_VAR
VAR
END_VAR

ptrData^ := ptrData^ AND NOT (SHR(DWORD#16#00008000,F_BACnet_BitFieldBit(bitNbr)));
F_BACnet_UnSetBitFieldBit := ptrData^;

END_FUNCTION

// POUs/Helper/Flags/F_BACnet_EventEnable
FUNCTION F_BACnet_EventEnable : UINT
VAR_INPUT
	stEvtEn       : ST_BA_EventTransitions;
END_VAR
VAR
	nEvtEnToFlt     : UINT;
	nEvtEnToNmal    : UINT;
	nEvtEnToOffnmal : UINT;
	nEvtEnNo        : UINT;
END_VAR

(*=============================================*)
(*EventEnable*)
IF	stEvtEn.bToFault
THEN
	nEvtEnToFlt := 16#4000;
ELSE
	nEvtEnToFlt := 16#0;
END_IF

IF	stEvtEn.bToNormal
THEN
	nEvtEnToNmal := 16#2000;
ELSE
	nEvtEnToNmal := 16#0;
END_IF

IF	stEvtEn.bToOffnormal
THEN
	nEvtEnToOffnmal := 16#8000;
ELSE
	nEvtEnToOffnmal := 16#0;
END_IF

nEvtEnNo := 5;

F_BACnet_EventEnable := nEvtEnNo + nEvtEnToFlt + nEvtEnToNmal + nEvtEnToOffnmal;
(*=============================================*)

END_FUNCTION

// POUs/Helper/Flags/F_BACnet_EventTransitionFlags
FUNCTION F_BACnet_EventTransitionFlags : ST_BA_EventTransitions
VAR_INPUT
	data	: WORD;
END_VAR
VAR
END_VAR

F_BACnet_EventTransitionFlags.bToNormal := F_BACnet_IsBitFieldBitSet(data, E_BACnet_EventTransitionBits.eToNormal);
F_BACnet_EventTransitionFlags.bToOffnormal := F_BACnet_IsBitFieldBitSet(data, E_BACnet_EventTransitionBits.eToOffnormal);
F_BACnet_EventTransitionFlags.bToFault := F_BACnet_IsBitFieldBitSet(data, E_BACnet_EventTransitionBits.eToFault);

END_FUNCTION

// POUs/Helper/Flags/F_BACnet_GetEventTransFlagsData
FUNCTION F_BACnet_GetEventTransFlagsData : WORD
VAR_INPUT
	Flags	: ST_BA_EventTransitions;
END_VAR
VAR
END_VAR

F_BACnet_GetEventTransFlagsData := 16#0005;
IF Flags.bToNormal THEN
	F_BACnet_GetEventTransFlagsData := DWORD_TO_WORD(F_BACnet_SetBitFieldBit(ptrData:=ADR(F_BACnet_GetEventTransFlagsData), bitNbr:=E_BACnet_EventTransitionBits.eToNormal));
END_IF
IF Flags.bToOffnormal THEN
	F_BACnet_GetEventTransFlagsData := DWORD_TO_WORD(F_BACnet_SetBitFieldBit(ptrData:=ADR(F_BACnet_GetEventTransFlagsData), bitNbr:=E_BACnet_EventTransitionBits.eToOffnormal));
END_IF
IF Flags.bToFault THEN
	F_BACnet_GetEventTransFlagsData := DWORD_TO_WORD(F_BACnet_SetBitFieldBit(ptrData:=ADR(F_BACnet_GetEventTransFlagsData), bitNbr:=E_BACnet_EventTransitionBits.eToFault));
END_IF

END_FUNCTION

// POUs/Helper/Flags/F_BACnet_GetLimitEnFlagsData
FUNCTION F_BACnet_GetLimitEnFlagsData : WORD
VAR_INPUT
	Flags	: ST_BACnet_LimitEnable;
END_VAR
VAR
END_VAR

F_BACnet_GetLimitEnFlagsData := 16#0006;
IF Flags.highLimitEnable THEN
	F_BACnet_GetLimitEnFlagsData := DWORD_TO_WORD(F_BACnet_SetBitFieldBit(ptrData:=ADR(F_BACnet_GetLimitEnFlagsData), bitNbr:=E_BACnet_LimitEnableBits.eHighLimit));
END_IF
IF Flags.lowLimitEnable THEN
	F_BACnet_GetLimitEnFlagsData := DWORD_TO_WORD(F_BACnet_SetBitFieldBit(ptrData:=ADR(F_BACnet_GetLimitEnFlagsData), bitNbr:=E_BACnet_LimitEnableBits.eLowLimit));
END_IF

END_FUNCTION

// POUs/Helper/Flags/F_BACnet_GetStatusFlagsData
FUNCTION F_BACnet_GetStatusFlagsData : WORD
VAR_INPUT
	Flags : ST_BA_StatusFlags;
END_VAR

F_BACnet_GetStatusFlagsData	:= 16#0004;
IF Flags.bInAlarm THEN
	F_BACnet_GetStatusFlagsData := DWORD_TO_WORD(F_BACnet_SetBitFieldBit(ptrData:=ADR(F_BACnet_GetStatusFlagsData), bitNbr:=E_BACnet_StatusFlags.eInAlarm));
END_IF
IF Flags.bFault THEN
	F_BACnet_GetStatusFlagsData := DWORD_TO_WORD(F_BACnet_SetBitFieldBit(ptrData:=ADR(F_BACnet_GetStatusFlagsData), bitNbr:=E_BACnet_StatusFlags.eFault));
END_IF
IF Flags.bOverridden THEN
	F_BACnet_GetStatusFlagsData := DWORD_TO_WORD(F_BACnet_SetBitFieldBit(ptrData:=ADR(F_BACnet_GetStatusFlagsData), bitNbr:=E_BACnet_StatusFlags.eOverridden));
END_IF
IF Flags.bOutOfService THEN
	F_BACnet_GetStatusFlagsData := DWORD_TO_WORD(F_BACnet_SetBitFieldBit(ptrData:=ADR(F_BACnet_GetStatusFlagsData), bitNbr:=E_BACnet_StatusFlags.eOutOfService));
END_IF

END_FUNCTION

// POUs/Helper/Flags/F_BACnet_LimitEnable
FUNCTION F_BACnet_LimitEnable : UINT
VAR_INPUT
	stLimEn         : ST_BACnet_LimitEnable;
END_VAR
VAR
	nHiLimEn     : UINT;
	nLowLimEn    : UINT;
	nLimEnNo     : UINT;
END_VAR

(*=============================================*)
IF	stLimEn.highLimitEnable
THEN
	nHiLimEn := 16#4000;
ELSE
	nHiLimEn := 16#0;
END_IF


IF	stLimEn.lowLimitEnable
THEN
	nLowLimEn := 16#8000;
ELSE
	nLowLimEn := 16#0;
END_IF

nLimEnNo := 16#6;

F_BACnet_LimitEnable := nLimEnNo + nHiLimEn + nLowLimEn;
(*=============================================*)

END_FUNCTION

// POUs/Helper/Flags/F_BACnet_LimitEnableFlags
FUNCTION F_BACnet_LimitEnableFlags : ST_BACnet_LimitEnable
VAR_INPUT
	data	: WORD;
END_VAR
VAR
END_VAR

F_BACnet_LimitEnableFlags.highLimitEnable := F_BACnet_IsBitFieldBitSet( data:=data, bitNbr:=E_BACnet_LimitEnableBits.eHighLimit);
F_BACnet_LimitEnableFlags.lowLimitEnable := F_BACnet_IsBitFieldBitSet( data:=data, bitNbr:=E_BACnet_LimitEnableBits.eLowLimit);

END_FUNCTION

// POUs/Helper/Flags/F_BACnet_StatusFlags
FUNCTION F_BACnet_StatusFlags : ST_BA_StatusFlags
VAR_INPUT
	data	: WORD;
END_VAR
VAR
END_VAR

F_BACnet_StatusFlags.bInAlarm:= F_BACnet_IsBitFieldBitSet( data:=data, bitNbr:=E_BACnet_StatusFlags.eInAlarm);
F_BACnet_StatusFlags.bFault:= F_BACnet_IsBitFieldBitSet( data:=data, bitNbr:=E_BACnet_StatusFlags.eFault);
F_BACnet_StatusFlags.bOverridden:= F_BACnet_IsBitFieldBitSet( data:=data, bitNbr:=E_BACnet_StatusFlags.eOverridden);
F_BACnet_StatusFlags.bOutOfService:= F_BACnet_IsBitFieldBitSet( data:=data, bitNbr:=E_BACnet_StatusFlags.eOutOfService);

END_FUNCTION

// POUs/Helper/MultiState/F_BACnet_EnMultiStatePV
FUNCTION F_BACnet_EnMultiStatePV : UDINT
VAR_INPUT
	bEnable			: BOOL;
	nValue			: UDINT;
END_VAR

IF (bEnable) THEN
	F_BACnet_EnMultiStatePV := MAX(nValue, E_BACnet_MultistateVal.eMin);
ELSE
	F_BACnet_EnMultiStatePV := E_BACnet_MultistateVal.eNull;
END_IF

END_FUNCTION

// POUs/Helper/MultiState/F_BACnet_MultiStatePV
FUNCTION F_BACnet_MultiStatePV : UDINT
VAR_INPUT
	bEnable						: BOOL; (* TRUE = commit to stack, FALSE = do-nothing *)
	bNull						: BOOL; (* TRUE = clear priority, FALSE = write number from state input *)
	nState						: UDINT; (* multi-state [1..max-number-of-states] *)
END_VAR

